Yaskawa INFORM job: DEMO_ROOF_UPPER_0625_3PAINT_26.JBI

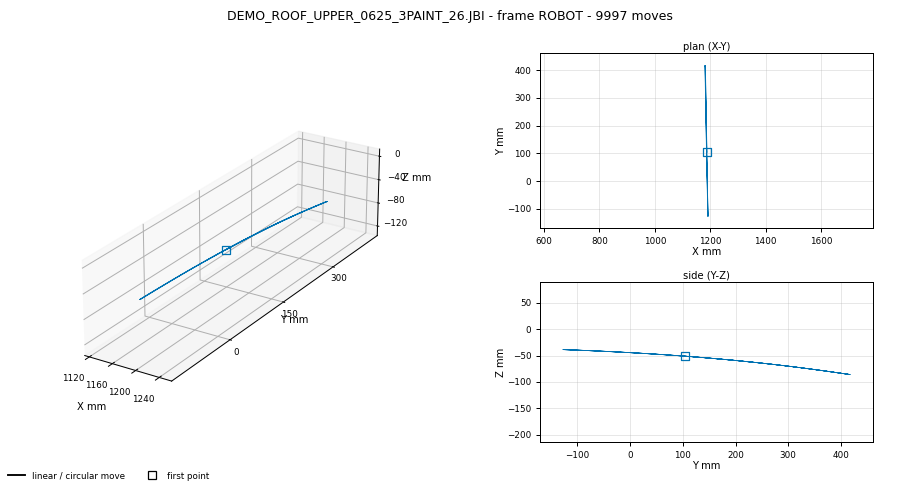
[picture p0: tool path of DEMO_ROOF_UPPER_0625_3PAINT_26.JBI in frame ROBOT, 9997 of 9997 moves have a stored position in this frame; points joined in program order, loops and branches not executed]
/JOB
//NAME DEMO_ROOF_UPPER_0625_3PAINT26
//POS
///NPOS 9997,0,0,0,0,0
///TOOL 0
///USER 0
///POSTYPE ROBOT
///RECTAN
///RCONF 1,0,0,0,0,0,0,0,0,0,0,0,0,0,0,0,0,0,0,0,0,0,0,0
C00000=1188.061,103.927,-51.027,-178.803,6.071,148.735
C00001=1188.057,104.176,-51.046,-178.800,6.072,148.734
C00002=1188.052,104.425,-51.064,-178.798,6.073,148.734
C00003=1188.047,104.675,-51.083,-178.795,6.075,148.733
C00004=1188.042,104.924,-51.102,-178.793,6.076,148.733
C00005=1188.036,105.173,-51.120,-178.790,6.077,148.732
C00006=1188.032,105.423,-51.139,-178.787,6.078,148.732
C00007=1188.027,105.672,-51.157,-178.785,6.080,148.731
C00008=1188.023,105.921,-51.177,-178.782,6.080,148.731
C00009=1188.018,106.171,-51.195,-178.779,6.082,148.730
C00010=1188.012,106.439,-51.216,-178.776,6.083,148.730
C00011=1188.008,106.708,-51.236,-178.774,6.084,148.729
C00012=1188.002,106.975,-51.256,-178.771,6.086,148.729
C00013=1187.996,107.244,-51.276,-178.768,6.087,148.728
C00014=1187.992,107.493,-51.295,-178.766,6.088,148.728
C00015=1187.987,107.743,-51.314,-178.763,6.090,148.727
C00016=1187.983,107.992,-51.333,-178.760,6.090,148.727
C00017=1187.978,108.241,-51.351,-178.758,6.092,148.726
C00018=1187.973,108.490,-51.370,-178.755,6.094,148.726
C00019=1187.969,108.739,-51.389,-178.752,6.094,148.725
C00020=1187.963,108.989,-51.408,-178.750,6.096,148.725
C00021=1187.959,109.238,-51.427,-178.747,6.097,148.724
C00022=1187.954,109.487,-51.446,-178.744,6.098,148.724
C00023=1187.949,109.736,-51.464,-178.742,6.099,148.723
C00024=1187.944,109.986,-51.484,-178.739,6.101,148.723
C00025=1187.939,110.234,-51.503,-178.737,6.102,148.722
C00026=1187.934,110.484,-51.521,-178.734,6.103,148.722
C00027=1187.929,110.733,-51.541,-178.731,6.105,148.721
C00028=1187.925,110.983,-51.560,-178.729,6.106,148.721
C00029=1187.919,111.232,-51.578,-178.726,6.107,148.720
C00030=1187.915,111.481,-51.597,-178.723,6.108,148.720
C00031=1187.910,111.730,-51.617,-178.721,6.110,148.719
C00032=1187.906,111.979,-51.636,-178.718,6.110,148.719
C00033=1187.900,112.229,-51.654,-178.715,6.112,148.718
C00034=1187.896,112.478,-51.673,-178.712,6.113,148.718
C00035=1187.891,112.727,-51.693,-178.710,6.114,148.717
C00036=1187.886,112.977,-51.712,-178.707,6.116,148.717
C00037=1187.881,113.226,-51.730,-178.705,6.117,148.716
C00038=1187.877,113.475,-51.750,-178.702,6.118,148.716
C00039=1187.871,113.724,-51.769,-178.700,6.119,148.715
C00040=1187.867,113.973,-51.788,-178.697,6.121,148.715
C00041=1187.862,114.222,-51.808,-178.694,6.122,148.714
C00042=1187.857,114.472,-51.826,-178.691,6.123,148.714
C00043=1187.852,114.721,-51.845,-178.689,6.125,148.713
C00044=1187.847,114.971,-51.865,-178.687,6.126,148.713
C00045=1187.843,115.219,-51.884,-178.683,6.127,148.712
C00046=1187.838,115.469,-51.903,-178.681,6.129,148.712
C00047=1187.833,115.718,-51.923,-178.679,6.130,148.712
C00048=1187.829,115.967,-51.942,-178.675,6.131,148.711
C00049=1187.823,116.216,-51.961,-178.673,6.132,148.710
C00050=1187.819,116.465,-51.981,-178.671,6.134,148.710
C00051=1187.813,116.714,-52.000,-178.667,6.135,148.709
C00052=1187.809,116.964,-52.018,-178.665,6.136,148.709
C00053=1187.804,117.214,-52.038,-178.663,6.138,148.709
C00054=1187.799,117.462,-52.057,-178.660,6.138,148.708
C00055=1187.795,117.712,-52.076,-178.657,6.140,148.708
C00056=1187.790,117.961,-52.096,-178.655,6.142,148.707
C00057=1187.785,118.210,-52.115,-178.652,6.142,148.707
C00058=1187.780,118.460,-52.135,-178.649,6.144,148.706
C00059=1187.775,118.708,-52.154,-178.647,6.145,148.706
C00060=1187.771,118.958,-52.173,-178.644,6.147,148.705
C00061=1187.765,119.207,-52.192,-178.641,6.148,148.705
C00062=1187.761,119.456,-52.212,-178.639,6.149,148.704
C00063=1187.756,119.706,-52.232,-178.636,6.151,148.704
C00064=1187.752,119.954,-52.251,-178.633,6.152,148.703
C00065=1187.747,120.203,-52.271,-178.631,6.153,148.703
C00066=1187.741,120.452,-52.290,-178.628,6.155,148.702
C00067=1187.737,120.702,-52.310,-178.626,6.156,148.702
C00068=1187.732,120.951,-52.329,-178.623,6.157,148.701
C00069=1187.727,121.200,-52.348,-178.620,6.159,148.701
C00070=1187.723,121.450,-52.368,-178.618,6.160,148.700
C00071=1187.718,121.699,-52.387,-178.615,6.161,148.700
C00072=1187.713,121.948,-52.407,-178.612,6.163,148.699
C00073=1187.708,122.197,-52.427,-178.610,6.164,148.699
C00074=1187.703,122.446,-52.447,-178.607,6.166,148.699
C00075=1187.698,122.695,-52.466,-178.604,6.166,148.698
C00076=1187.694,122.945,-52.485,-178.602,6.168,148.698
C00077=1187.689,123.194,-52.505,-178.599,6.170,148.697
C00078=1187.684,123.443,-52.524,-178.596,6.170,148.697
C00079=1187.680,123.692,-52.544,-178.594,6.172,148.696
C00080=1187.675,123.942,-52.564,-178.591,6.174,148.696
C00081=1187.669,124.190,-52.583,-178.588,6.174,148.695
C00082=1187.665,124.440,-52.603,-178.586,6.176,148.695
C00083=1187.660,124.689,-52.623,-178.583,6.178,148.694
C00084=1187.655,124.938,-52.643,-178.581,6.179,148.694
C00085=1187.650,125.187,-52.662,-178.578,6.180,148.693
C00086=1187.646,125.437,-52.681,-178.575,6.182,148.693
C00087=1187.642,125.686,-52.702,-178.573,6.183,148.692
C00088=1187.636,125.934,-52.721,-178.570,6.184,148.692
C00089=1187.632,126.184,-52.741,-178.567,6.186,148.691
C00090=1187.627,126.433,-52.761,-178.565,6.187,148.691
C00091=1187.622,126.683,-52.781,-178.562,6.188,148.690
C00092=1187.617,126.931,-52.800,-178.559,6.190,148.690
C00093=1187.613,127.180,-52.820,-178.557,6.191,148.690
C00094=1187.608,127.430,-52.840,-178.554,6.193,148.689
C00095=1187.603,127.679,-52.860,-178.551,6.194,148.689
C00096=1187.598,127.928,-52.880,-178.549,6.195,148.688
C00097=1187.593,128.177,-52.899,-178.546,6.197,148.688
C00098=1187.589,128.426,-52.920,-178.543,6.198,148.687
C00099=1187.584,128.676,-52.939,-178.541,6.199,148.687
C00100=1187.579,128.924,-52.959,-178.538,6.201,148.686
C00101=1187.574,129.174,-52.979,-178.536,6.203,148.686
C00102=1187.570,129.423,-52.999,-178.533,6.203,148.685
C00103=1187.565,129.672,-53.020,-178.530,6.205,148.685
C00104=1187.560,129.922,-53.039,-178.528,6.207,148.685
C00105=1187.555,130.170,-53.059,-178.525,6.208,148.684
C00106=1187.550,130.420,-53.079,-178.522,6.209,148.684
C00107=1187.546,130.669,-53.099,-178.520,6.211,148.683
C00108=1187.541,130.918,-53.119,-178.517,6.213,148.683
C00109=1187.536,131.167,-53.139,-178.514,6.213,148.682
C00110=1187.531,131.416,-53.159,-178.512,6.215,148.682
C00111=1187.527,131.665,-53.179,-178.509,6.217,148.681
C00112=1187.522,131.915,-53.199,-178.507,6.218,148.681
C00113=1187.517,132.164,-53.220,-178.504,6.219,148.680
C00114=1187.512,132.433,-53.241,-178.501,6.221,148.680
C00115=1187.506,132.701,-53.263,-178.498,6.223,148.680
C00116=1187.502,132.970,-53.284,-178.495,6.224,148.679
C00117=1187.496,133.238,-53.307,-178.492,6.226,148.679
C00118=1187.491,133.488,-53.326,-178.490,6.226,148.678
C00119=1187.487,133.736,-53.347,-178.487,6.228,148.678
C00120=1187.482,133.986,-53.366,-178.484,6.230,148.677
C00121=1187.478,134.235,-53.387,-178.482,6.232,148.677
C00122=1187.472,134.484,-53.407,-178.479,6.232,148.676
C00123=1187.467,134.733,-53.427,-178.476,6.234,148.676
C00124=1187.463,134.982,-53.447,-178.474,6.236,148.675
C00125=1187.458,135.231,-53.468,-178.472,6.237,148.675
C00126=1187.454,135.480,-53.488,-178.468,6.238,148.674
C00127=1187.448,135.730,-53.508,-178.466,6.240,148.674
C00128=1187.444,135.979,-53.529,-178.463,6.242,148.674
C00129=1187.440,136.228,-53.549,-178.461,6.242,148.673
C00130=1187.435,136.477,-53.569,-178.458,6.244,148.673
C00131=1187.430,136.727,-53.590,-178.455,6.246,148.672
C00132=1187.425,136.976,-53.610,-178.452,6.247,148.672
C00133=1187.420,137.224,-53.630,-178.450,6.248,148.671
C00134=1187.415,137.473,-53.650,-178.447,6.250,148.671
C00135=1187.410,137.723,-53.671,-178.444,6.252,148.670
C00136=1187.406,137.972,-53.691,-178.442,6.252,148.670
C00137=1187.401,138.220,-53.712,-178.440,6.254,148.670
C00138=1187.396,138.470,-53.732,-178.437,6.256,148.669
C00139=1187.392,138.719,-53.753,-178.434,6.257,148.669
C00140=1187.387,138.968,-53.773,-178.432,6.258,148.668
C00141=1187.382,139.218,-53.793,-178.429,6.260,148.668
C00142=1187.377,139.466,-53.814,-178.426,6.262,148.667
C00143=1187.373,139.715,-53.834,-178.423,6.264,148.667
C00144=1187.368,139.965,-53.855,-178.421,6.264,148.666
C00145=1187.363,140.214,-53.876,-178.418,6.266,148.666
C00146=1187.359,140.463,-53.896,-178.415,6.268,148.666
C00147=1187.354,140.712,-53.917,-178.413,6.270,148.665
C00148=1187.349,140.961,-53.937,-178.410,6.271,148.665
C00149=1187.344,141.211,-53.958,-178.407,6.272,148.664
C00150=1187.339,141.460,-53.978,-178.405,6.274,148.664
C00151=1187.335,141.709,-53.998,-178.402,6.275,148.664
C00152=1187.330,141.958,-54.019,-178.399,6.277,148.663
C00153=1187.325,142.207,-54.040,-178.397,6.278,148.663
C00154=1187.320,142.456,-54.061,-178.394,6.280,148.662
C00155=1187.316,142.705,-54.081,-178.391,6.281,148.662
C00156=1187.311,142.954,-54.101,-178.389,6.283,148.661
C00157=1187.306,143.203,-54.122,-178.387,6.284,148.661
C00158=1187.302,143.452,-54.143,-178.384,6.286,148.661
C00159=1187.297,143.701,-54.164,-178.381,6.287,148.660
C00160=1187.292,143.950,-54.184,-178.378,6.289,148.660
C00161=1187.287,144.199,-54.206,-178.375,6.291,148.659
C00162=1187.283,144.448,-54.226,-178.373,6.292,148.659
C00163=1187.278,144.697,-54.247,-178.371,6.293,148.658
C00164=1187.274,144.947,-54.268,-178.367,6.295,148.658
C00165=1187.269,145.196,-54.289,-178.365,6.297,148.657
C00166=1187.264,145.445,-54.309,-178.363,6.298,148.657
C00167=1187.259,145.694,-54.330,-178.360,6.299,148.657
C00168=1187.255,145.943,-54.350,-178.357,6.301,148.656
C00169=1187.249,146.193,-54.371,-178.355,6.303,148.656
C00170=1187.245,146.441,-54.392,-178.351,6.304,148.655
C00171=1187.240,146.690,-54.413,-178.349,6.305,148.655
C00172=1187.236,146.939,-54.434,-178.347,6.307,148.655
C00173=1187.230,147.188,-54.455,-178.344,6.309,148.654
C00174=1187.225,147.438,-54.476,-178.341,6.310,148.654
C00175=1187.222,147.687,-54.497,-178.339,6.312,148.653
C00176=1187.217,147.936,-54.518,-178.335,6.314,148.653
C00177=1187.212,148.185,-54.539,-178.333,6.315,148.652
C00178=1187.207,148.434,-54.560,-178.331,6.316,148.652
C00179=1187.203,148.682,-54.581,-178.328,6.318,148.652
C00180=1187.198,148.932,-54.602,-178.325,6.320,148.651
C00181=1187.193,149.181,-54.623,-178.322,6.322,148.651
C00182=1187.189,149.431,-54.643,-178.320,6.322,148.650
C00183=1187.184,149.679,-54.665,-178.317,6.324,148.650
C00184=1187.179,149.928,-54.686,-178.315,6.326,148.649
C00185=1187.174,150.177,-54.706,-178.312,6.328,148.649
C00186=1187.169,150.426,-54.728,-178.309,6.329,148.649
C00187=1187.164,150.675,-54.749,-178.306,6.331,148.648
C00188=1187.160,150.925,-54.770,-178.304,6.332,148.648
C00189=1187.155,151.174,-54.791,-178.301,6.334,148.647
C00190=1187.150,151.423,-54.812,-178.299,6.335,148.647
C00191=1187.146,151.672,-54.833,-178.296,6.337,148.647
C00192=1187.141,151.920,-54.854,-178.293,6.339,148.646
C00193=1187.136,152.170,-54.875,-178.291,6.340,148.646
C00194=1187.132,152.419,-54.897,-178.288,6.342,148.645
C00195=1187.127,152.668,-54.918,-178.286,6.343,148.645
C00196=1187.122,152.917,-54.939,-178.283,6.345,148.645
C00197=1187.117,153.166,-54.960,-178.280,6.347,148.644
C00198=1187.113,153.416,-54.981,-178.277,6.348,148.644
C00199=1187.108,153.664,-55.003,-178.274,6.350,148.643
C00200=1187.103,153.913,-55.024,-178.272,6.351,148.643
C00201=1187.098,154.162,-55.045,-178.270,6.353,148.643
C00202=1187.094,154.411,-55.066,-178.267,6.355,148.642
C00203=1187.090,154.660,-55.088,-178.264,6.356,148.642
C00204=1187.084,154.910,-55.109,-178.262,6.358,148.641
C00205=1187.080,155.158,-55.131,-178.258,6.360,148.641
C00206=1187.074,155.408,-55.152,-178.256,6.361,148.640
C00207=1187.071,155.657,-55.173,-178.254,6.362,148.640
C00208=1187.066,155.906,-55.194,-178.251,6.364,148.640
C00209=1187.061,156.154,-55.216,-178.248,6.366,148.639
C00210=1187.057,156.404,-55.238,-178.246,6.368,148.639
C00211=1187.051,156.653,-55.259,-178.243,6.369,148.639
C00212=1187.046,156.902,-55.280,-178.240,6.371,148.638
C00213=1187.042,157.151,-55.301,-178.238,6.373,148.638
C00214=1187.038,157.400,-55.323,-178.235,6.373,148.637
C00215=1187.033,157.649,-55.344,-178.232,6.375,148.637
C00216=1187.028,157.898,-55.365,-178.230,6.377,148.636
C00217=1187.023,158.147,-55.387,-178.227,6.379,148.636
C00218=1187.019,158.416,-55.410,-178.224,6.381,148.636
C00219=1187.013,158.684,-55.434,-178.222,6.382,148.635
C00220=1187.008,158.953,-55.457,-178.218,6.384,148.635
C00221=1187.003,159.223,-55.480,-178.215,6.386,148.634
C00222=1186.998,159.472,-55.502,-178.213,6.387,148.634
C00223=1186.994,159.721,-55.524,-178.210,6.389,148.634
C00224=1186.988,159.970,-55.545,-178.208,6.391,148.633
C00225=1186.984,160.219,-55.567,-178.205,6.393,148.633
C00226=1186.979,160.468,-55.588,-178.202,6.394,148.633
C00227=1186.975,160.716,-55.610,-178.200,6.396,148.632
C00228=1186.971,160.966,-55.631,-178.197,6.398,148.632
C00229=1186.966,161.215,-55.653,-178.194,6.400,148.631
C00230=1186.961,161.464,-55.675,-178.191,6.401,148.631
C00231=1186.957,161.713,-55.696,-178.189,6.402,148.630
C00232=1186.952,161.962,-55.718,-178.186,6.404,148.630
C00233=1186.947,162.211,-55.739,-178.184,6.406,148.630
C00234=1186.942,162.460,-55.761,-178.181,6.407,148.629
C00235=1186.938,162.709,-55.783,-178.178,6.409,148.629
C00236=1186.933,162.958,-55.805,-178.176,6.411,148.629
C00237=1186.928,163.207,-55.826,-178.173,6.413,148.628
C00238=1186.924,163.456,-55.848,-178.170,6.415,148.628
C00239=1186.919,163.705,-55.870,-178.168,6.416,148.627
C00240=1186.915,163.954,-55.892,-178.165,6.418,148.627
C00241=1186.909,164.204,-55.914,-178.162,6.420,148.627
C00242=1186.904,164.452,-55.935,-178.159,6.422,148.626
C00243=1186.900,164.702,-55.957,-178.157,6.423,148.626
C00244=1186.895,164.950,-55.979,-178.155,6.424,148.626
C00245=1186.891,165.200,-56.001,-178.152,6.426,148.625
C00246=1186.886,165.448,-56.023,-178.149,6.428,148.625
C00247=1186.881,165.698,-56.045,-178.146,6.429,148.624
C00248=1186.877,165.946,-56.067,-178.144,6.431,148.624
C00249=1186.872,166.196,-56.089,-178.141,6.433,148.624
C00250=1186.867,166.444,-56.110,-178.138,6.435,148.623
C00251=1186.863,166.694,-56.132,-178.135,6.437,148.623
C00252=1186.858,166.942,-56.155,-178.133,6.438,148.622
C00253=1186.853,167.191,-56.176,-178.130,6.440,148.622
C00254=1186.848,167.440,-56.198,-178.127,6.442,148.622
C00255=1186.844,167.688,-56.221,-178.125,6.444,148.621
C00256=1186.840,167.938,-56.243,-178.122,6.445,148.621
C00257=1186.835,168.186,-56.265,-178.119,6.447,148.621
C00258=1186.830,168.436,-56.287,-178.117,6.448,148.620
C00259=1186.825,168.685,-56.309,-178.115,6.450,148.620
C00260=1186.821,168.934,-56.331,-178.112,6.452,148.619
C00261=1186.816,169.183,-56.353,-178.109,6.453,148.619
C00262=1186.812,169.432,-56.375,-178.107,6.455,148.619
C00263=1186.806,169.681,-56.397,-178.104,6.457,148.618
C00264=1186.802,169.930,-56.420,-178.101,6.459,148.618
C00265=1186.798,170.179,-56.442,-178.099,6.461,148.618
C00266=1186.793,170.428,-56.463,-178.096,6.462,148.617
C00267=1186.788,170.677,-56.486,-178.093,6.464,148.617
C00268=1186.783,170.926,-56.508,-178.091,6.466,148.617
C00269=1186.779,171.175,-56.531,-178.088,6.468,148.616
C00270=1186.774,171.423,-56.552,-178.085,6.470,148.616
C00271=1186.769,171.673,-56.575,-178.083,6.471,148.615
C00272=1186.764,171.922,-56.597,-178.080,6.473,148.615
C00273=1186.760,172.170,-56.619,-178.077,6.475,148.615
C00274=1186.755,172.420,-56.642,-178.074,6.477,148.614
C00275=1186.750,172.669,-56.664,-178.072,6.478,148.614
C00276=1186.746,172.917,-56.686,-178.069,6.480,148.614
C00277=1186.742,173.166,-56.708,-178.066,6.482,148.613
C00278=1186.737,173.416,-56.731,-178.064,6.484,148.613
C00279=1186.732,173.664,-56.753,-178.061,6.486,148.613
C00280=1186.728,173.913,-56.775,-178.058,6.487,148.612
C00281=1186.723,174.163,-56.798,-178.056,6.489,148.612
C00282=1186.718,174.411,-56.820,-178.053,6.491,148.611
C00283=1186.713,174.660,-56.843,-178.050,6.493,148.611
C00284=1186.709,174.910,-56.865,-178.048,6.494,148.611
C00285=1186.704,175.158,-56.887,-178.045,6.496,148.610
C00286=1186.699,175.407,-56.910,-178.042,6.498,148.610
C00287=1186.695,175.655,-56.932,-178.040,6.500,148.610
C00288=1186.690,175.905,-56.954,-178.037,6.502,148.609
C00289=1186.685,176.154,-56.977,-178.034,6.503,148.609
C00290=1186.681,176.402,-56.999,-178.032,6.505,148.609
C00291=1186.676,176.652,-57.022,-178.029,6.507,148.608
C00292=1186.672,176.901,-57.045,-178.026,6.509,148.608
C00293=1186.666,177.150,-57.067,-178.024,6.511,148.607
C00294=1186.662,177.398,-57.090,-178.021,6.512,148.607
C00295=1186.657,177.648,-57.112,-178.018,6.514,148.607
C00296=1186.653,177.896,-57.135,-178.016,6.516,148.606
C00297=1186.649,178.145,-57.157,-178.013,6.518,148.606
C00298=1186.644,178.395,-57.180,-178.010,6.519,148.606
C00299=1186.639,178.643,-57.203,-178.008,6.522,148.606
C00300=1186.634,178.892,-57.225,-178.005,6.523,148.605
C00301=1186.630,179.141,-57.248,-178.003,6.525,148.605
C00302=1186.625,179.391,-57.271,-178.000,6.527,148.604
C00303=1186.621,179.639,-57.293,-177.997,6.529,148.604
C00304=1186.616,179.888,-57.317,-177.995,6.531,148.604
C00305=1186.612,180.137,-57.339,-177.992,6.532,148.603
C00306=1186.606,180.385,-57.362,-177.989,6.534,148.603
C00307=1186.602,180.635,-57.384,-177.987,6.536,148.603
C00308=1186.597,180.884,-57.407,-177.984,6.538,148.602
C00309=1186.593,181.133,-57.430,-177.981,6.539,148.602
C00310=1186.588,181.381,-57.452,-177.979,6.541,148.602
C00311=1186.583,181.630,-57.475,-177.976,6.543,148.601
C00312=1186.579,181.879,-57.498,-177.973,6.545,148.601
C00313=1186.575,182.128,-57.521,-177.971,6.547,148.600
C00314=1186.570,182.377,-57.543,-177.968,6.548,148.600
C00315=1186.565,182.626,-57.567,-177.965,6.550,148.600
C00316=1186.560,182.875,-57.590,-177.963,6.552,148.600
C00317=1186.556,183.124,-57.613,-177.961,6.554,148.599
C00318=1186.551,183.373,-57.635,-177.958,6.556,148.599
C00319=1186.546,183.622,-57.658,-177.955,6.558,148.599
C00320=1186.542,183.870,-57.681,-177.952,6.560,148.598
C00321=1186.537,184.119,-57.704,-177.949,6.562,148.598
C00322=1186.533,184.389,-57.729,-177.947,6.564,148.598
C00323=1186.527,184.659,-57.754,-177.944,6.566,148.597
C00324=1186.522,184.928,-57.779,-177.941,6.568,148.597
C00325=1186.518,185.198,-57.803,-177.938,6.570,148.596
C00326=1186.513,185.447,-57.827,-177.935,6.572,148.596
C00327=1186.508,185.696,-57.850,-177.933,6.574,148.596
C00328=1186.504,185.945,-57.873,-177.930,6.575,148.595
C00329=1186.499,186.193,-57.896,-177.927,6.577,148.595
C00330=1186.494,186.443,-57.918,-177.925,6.579,148.595
C00331=1186.489,186.692,-57.942,-177.922,6.581,148.594
C00332=1186.485,186.940,-57.965,-177.919,6.583,148.594
C00333=1186.481,187.189,-57.988,-177.917,6.584,148.594
C00334=1186.476,187.438,-58.011,-177.914,6.587,148.594
C00335=1186.471,187.687,-58.034,-177.911,6.589,148.593
C00336=1186.467,187.935,-58.057,-177.909,6.591,148.593
C00337=1186.462,188.184,-58.080,-177.906,6.593,148.592
C00338=1186.457,188.433,-58.104,-177.903,6.595,148.592
C00339=1186.452,188.682,-58.127,-177.901,6.596,148.592
C00340=1186.449,188.931,-58.150,-177.898,6.598,148.591
C00341=1186.444,189.180,-58.173,-177.895,6.600,148.591
C00342=1186.439,189.429,-58.197,-177.893,6.602,148.591
C00343=1186.434,189.678,-58.220,-177.890,6.604,148.591
C00344=1186.429,189.927,-58.243,-177.888,6.606,148.590
C00345=1186.424,190.176,-58.266,-177.885,6.607,148.590
C00346=1186.420,190.424,-58.289,-177.882,6.610,148.590
C00347=1186.416,190.673,-58.313,-177.879,6.612,148.589
C00348=1186.411,190.922,-58.337,-177.877,6.614,148.589
C00349=1186.407,191.171,-58.360,-177.874,6.615,148.588
C00350=1186.402,191.420,-58.383,-177.872,6.618,148.588
C00351=1186.397,191.669,-58.407,-177.869,6.619,148.588
C00352=1186.393,191.918,-58.430,-177.866,6.621,148.588
C00353=1186.388,192.167,-58.453,-177.864,6.623,148.587
C00354=1186.384,192.415,-58.477,-177.861,6.625,148.587
C00355=1186.379,192.664,-58.500,-177.858,6.627,148.587
C00356=1186.375,192.913,-58.524,-177.855,6.629,148.586
C00357=1186.370,193.162,-58.547,-177.853,6.631,148.586
C00358=1186.365,193.411,-58.570,-177.850,6.633,148.586
C00359=1186.361,193.660,-58.594,-177.848,6.635,148.585
C00360=1186.356,193.909,-58.618,-177.845,6.637,148.585
C00361=1186.352,194.158,-58.641,-177.842,6.638,148.585
C00362=1186.347,194.407,-58.664,-177.840,6.640,148.584
C00363=1186.343,194.655,-58.688,-177.836,6.643,148.584
C00364=1186.338,194.904,-58.712,-177.834,6.645,148.584
C00365=1186.333,195.153,-58.735,-177.832,6.647,148.584
C00366=1186.329,195.402,-58.759,-177.829,6.649,148.583
C00367=1186.324,195.651,-58.783,-177.826,6.650,148.583
C00368=1186.319,195.900,-58.806,-177.824,6.652,148.583
C00369=1186.315,196.148,-58.830,-177.821,6.654,148.582
C00370=1186.310,196.397,-58.853,-177.819,6.656,148.582
C00371=1186.306,196.646,-58.877,-177.815,6.659,148.582
C00372=1186.301,196.895,-58.901,-177.813,6.661,148.581
C00373=1186.296,197.144,-58.924,-177.810,6.662,148.581
C00374=1186.292,197.392,-58.948,-177.807,6.664,148.581
C00375=1186.287,197.641,-58.972,-177.805,6.666,148.581
C00376=1186.283,197.890,-58.995,-177.803,6.668,148.580
C00377=1186.278,198.138,-59.019,-177.800,6.670,148.580
C00378=1186.274,198.388,-59.042,-177.797,6.672,148.580
C00379=1186.269,198.636,-59.067,-177.794,6.674,148.579
C00380=1186.264,198.885,-59.090,-177.791,6.676,148.579
C00381=1186.259,199.134,-59.115,-177.789,6.678,148.579
C00382=1186.255,199.383,-59.138,-177.787,6.680,148.578
C00383=1186.250,199.631,-59.162,-177.784,6.682,148.578
C00384=1186.246,199.881,-59.186,-177.781,6.684,148.578
C00385=1186.242,200.129,-59.210,-177.778,6.686,148.577
C00386=1186.237,200.378,-59.233,-177.776,6.688,148.577
C00387=1186.233,200.627,-59.257,-177.773,6.690,148.577
C00388=1186.227,200.876,-59.281,-177.770,6.692,148.577
C00389=1186.223,201.124,-59.305,-177.768,6.694,148.576
C00390=1186.218,201.373,-59.329,-177.765,6.696,148.576
C00391=1186.214,201.622,-59.353,-177.762,6.699,148.576
C00392=1186.210,201.871,-59.377,-177.760,6.700,148.575
C00393=1186.204,202.120,-59.401,-177.757,6.702,148.575
C00394=1186.200,202.369,-59.425,-177.754,6.704,148.575
C00395=1186.196,202.617,-59.449,-177.752,6.707,148.575
C00396=1186.191,202.866,-59.473,-177.749,6.709,148.574
C00397=1186.187,203.115,-59.497,-177.746,6.711,148.574
C00398=1186.181,203.363,-59.521,-177.744,6.712,148.574
C00399=1186.177,203.613,-59.545,-177.741,6.714,148.573
C00400=1186.173,203.862,-59.569,-177.739,6.716,148.573
C00401=1186.169,204.110,-59.593,-177.736,6.719,148.573
C00402=1186.163,204.359,-59.618,-177.733,6.721,148.573
C00403=1186.159,204.608,-59.641,-177.730,6.722,148.572
C00404=1186.155,204.857,-59.666,-177.728,6.725,148.572
C00405=1186.151,205.105,-59.690,-177.725,6.726,148.572
C00406=1186.145,205.354,-59.714,-177.722,6.729,148.571
C00407=1186.141,205.603,-59.738,-177.720,6.731,148.571
C00408=1186.136,205.851,-59.762,-177.717,6.733,148.571
C00409=1186.132,206.101,-59.787,-177.715,6.735,148.571
C00410=1186.127,206.349,-59.811,-177.712,6.737,148.570
C00411=1186.123,206.598,-59.835,-177.709,6.739,148.570
C00412=1186.118,206.847,-59.859,-177.707,6.741,148.570
C00413=1186.114,207.096,-59.883,-177.704,6.743,148.569
C00414=1186.109,207.345,-59.907,-177.701,6.745,148.569
C00415=1186.104,207.593,-59.932,-177.698,6.748,148.569
C00416=1186.100,207.842,-59.956,-177.696,6.750,148.569
C00417=1186.095,208.091,-59.981,-177.693,6.752,148.568
C00418=1186.091,208.339,-60.005,-177.691,6.753,148.568
C00419=1186.087,208.588,-60.029,-177.688,6.755,148.568
C00420=1186.081,208.837,-60.054,-177.685,6.758,148.568
C00421=1186.078,209.086,-60.079,-177.683,6.760,148.567
C00422=1186.072,209.335,-60.102,-177.680,6.762,148.567
C00423=1186.068,209.583,-60.127,-177.677,6.764,148.567
C00424=1186.063,209.832,-60.151,-177.674,6.766,148.566
C00425=1186.059,210.081,-60.176,-177.672,6.768,148.566
C00426=1186.054,210.351,-60.202,-177.669,6.770,148.566
C00427=1186.049,210.622,-60.229,-177.666,6.773,148.565
C00428=1186.044,210.893,-60.256,-177.663,6.775,148.565
C00429=1186.040,211.162,-60.282,-177.660,6.777,148.565
C00430=1186.034,211.411,-60.307,-177.658,6.779,148.565
C00431=1186.030,211.660,-60.331,-177.655,6.781,148.564
C00432=1186.026,211.909,-60.356,-177.652,6.784,148.564
C00433=1186.021,212.157,-60.380,-177.650,6.786,148.564
C00434=1186.016,212.406,-60.405,-177.647,6.788,148.564
C00435=1186.011,212.656,-60.430,-177.645,6.789,148.563
C00436=1186.007,212.904,-60.454,-177.641,6.792,148.563
C00437=1186.003,213.153,-60.479,-177.639,6.794,148.563
C00438=1185.998,213.401,-60.504,-177.636,6.796,148.563
C00439=1185.993,213.650,-60.528,-177.634,6.798,148.562
C00440=1185.990,213.899,-60.553,-177.631,6.801,148.562
C00441=1185.984,214.148,-60.578,-177.628,6.803,148.562
C00442=1185.980,214.396,-60.602,-177.626,6.804,148.561
C00443=1185.976,214.645,-60.627,-177.624,6.807,148.561
C00444=1185.971,214.894,-60.652,-177.620,6.809,148.561
C00445=1185.967,215.143,-60.676,-177.618,6.811,148.561
C00446=1185.962,215.391,-60.701,-177.616,6.813,148.561
C00447=1185.958,215.639,-60.726,-177.612,6.816,148.560
C00448=1185.953,215.889,-60.751,-177.610,6.818,148.560
C00449=1185.948,216.137,-60.776,-177.607,6.819,148.560
C00450=1185.944,216.387,-60.800,-177.605,6.822,148.559
C00451=1185.939,216.635,-60.825,-177.602,6.824,148.559
C00452=1185.934,216.883,-60.850,-177.599,6.826,148.559
C00453=1185.930,217.132,-60.875,-177.597,6.828,148.559
C00454=1185.926,217.381,-60.900,-177.594,6.831,148.558
C00455=1185.921,217.630,-60.925,-177.591,6.833,148.558
C00456=1185.917,217.878,-60.949,-177.589,6.835,148.558
C00457=1185.912,218.127,-60.975,-177.586,6.837,148.558
C00458=1185.907,218.376,-60.999,-177.583,6.839,148.557
C00459=1185.904,218.625,-61.024,-177.581,6.841,148.557
C00460=1185.899,218.873,-61.049,-177.578,6.843,148.557
C00461=1185.894,219.123,-61.074,-177.575,6.846,148.557
C00462=1185.889,219.371,-61.100,-177.573,6.848,148.556
C00463=1185.885,219.619,-61.124,-177.570,6.850,148.556
C00464=1185.881,219.868,-61.150,-177.568,6.852,148.556
C00465=1185.876,220.117,-61.174,-177.565,6.855,148.556
C00466=1185.871,220.365,-61.200,-177.562,6.856,148.555
C00467=1185.867,220.614,-61.224,-177.560,6.858,148.555
C00468=1185.863,220.863,-61.250,-177.557,6.861,148.555
C00469=1185.858,221.111,-61.274,-177.554,6.863,148.555
C00470=1185.853,221.360,-61.300,-177.552,6.865,148.555
C00471=1185.850,221.609,-61.325,-177.548,6.868,148.554
C00472=1185.845,221.857,-61.350,-177.546,6.870,148.554
C00473=1185.840,222.107,-61.375,-177.544,6.872,148.554
C00474=1185.835,222.355,-61.400,-177.541,6.873,148.553
C00475=1185.831,222.604,-61.425,-177.538,6.876,148.553
C00476=1185.826,222.852,-61.451,-177.536,6.878,148.553
C00477=1185.822,223.101,-61.477,-177.533,6.880,148.553
C00478=1185.817,223.350,-61.501,-177.530,6.883,148.553
C00479=1185.813,223.598,-61.526,-177.528,6.885,148.552
C00480=1185.808,223.847,-61.552,-177.525,6.887,148.552
C00481=1185.804,224.096,-61.577,-177.522,6.890,148.552
C00482=1185.800,224.345,-61.603,-177.520,6.891,148.552
C00483=1185.795,224.593,-61.628,-177.517,6.894,148.551
C00484=1185.790,224.842,-61.653,-177.514,6.896,148.551
C00485=1185.785,225.090,-61.678,-177.511,6.898,148.551
C00486=1185.781,225.339,-61.704,-177.509,6.900,148.551
C00487=1185.777,225.588,-61.728,-177.506,6.903,148.550
C00488=1185.773,225.836,-61.754,-177.504,6.905,148.550
C00489=1185.768,226.085,-61.780,-177.501,6.907,148.550
C00490=1185.764,226.333,-61.805,-177.498,6.910,148.550
C00491=1185.759,226.583,-61.830,-177.496,6.912,148.550
C00492=1185.755,226.832,-61.856,-177.493,6.913,148.549
C00493=1185.750,227.080,-61.881,-177.490,6.916,148.549
C00494=1185.746,227.329,-61.907,-177.488,6.918,148.549
C00495=1185.741,227.577,-61.932,-177.486,6.920,148.549
C00496=1185.736,227.826,-61.957,-177.482,6.923,148.548
C00497=1185.732,228.075,-61.983,-177.480,6.925,148.548
C00498=1185.727,228.323,-62.009,-177.478,6.927,148.548
C00499=1185.723,228.572,-62.034,-177.474,6.930,148.548
C00500=1185.719,228.821,-62.060,-177.472,6.932,148.548
C00501=1185.714,229.069,-62.085,-177.469,6.934,148.547
C00502=1185.710,229.317,-62.111,-177.467,6.937,148.547
C00503=1185.706,229.566,-62.137,-177.464,6.938,148.547
C00504=1185.700,229.815,-62.163,-177.461,6.941,148.547
C00505=1185.696,230.064,-62.188,-177.459,6.943,148.546
C00506=1185.691,230.313,-62.214,-177.456,6.945,148.546
C00507=1185.686,230.561,-62.239,-177.453,6.948,148.546
C00508=1185.682,230.810,-62.265,-177.451,6.950,148.546
C00509=1185.678,231.059,-62.291,-177.449,6.952,148.546
C00510=1185.674,231.307,-62.316,-177.445,6.955,148.545
C00511=1185.669,231.556,-62.342,-177.443,6.957,148.545
C00512=1185.665,231.804,-62.368,-177.440,6.959,148.545
C00513=1185.661,232.053,-62.393,-177.438,6.961,148.545
C00514=1185.655,232.302,-62.419,-177.435,6.963,148.544
C00515=1185.651,232.550,-62.446,-177.432,6.966,148.544
C00516=1185.647,232.799,-62.471,-177.430,6.968,148.544
C00517=1185.643,233.047,-62.497,-177.428,6.970,148.544
C00518=1185.638,233.295,-62.523,-177.424,6.973,148.544
C00519=1185.634,233.544,-62.548,-177.422,6.975,148.544
C00520=1185.629,233.793,-62.575,-177.419,6.978,148.543
C00521=1185.624,234.042,-62.600,-177.417,6.980,148.543
C00522=1185.620,234.290,-62.626,-177.414,6.982,148.543
C00523=1185.615,234.539,-62.652,-177.411,6.985,148.543
C00524=1185.611,234.788,-62.679,-177.409,6.986,148.542
C00525=1185.606,235.036,-62.704,-177.406,6.989,148.542
C00526=1185.602,235.285,-62.730,-177.403,6.991,148.542
C00527=1185.597,235.533,-62.756,-177.401,6.993,148.542
C00528=1185.593,235.782,-62.781,-177.398,6.996,148.542
C00529=1185.589,236.031,-62.808,-177.396,6.998,148.542
C00530=1185.584,236.302,-62.836,-177.393,7.001,148.541
C00531=1185.579,236.573,-62.865,-177.389,7.003,148.541
C00532=1185.573,236.845,-62.893,-177.387,7.006,148.541
C00533=1185.569,237.117,-62.921,-177.384,7.008,148.541
C00534=1185.565,237.365,-62.948,-177.382,7.010,148.541
C00535=1185.561,237.614,-62.974,-177.379,7.013,148.540
C00536=1185.556,237.863,-63.000,-177.377,7.015,148.540
C00537=1185.551,238.111,-63.026,-177.373,7.018,148.540
C00538=1185.547,238.360,-63.052,-177.371,7.020,148.540
C00539=1185.542,238.609,-63.078,-177.368,7.023,148.539
C00540=1185.538,238.857,-63.105,-177.366,7.025,148.539
C00541=1185.534,239.106,-63.130,-177.363,7.027,148.539
C00542=1185.529,239.354,-63.158,-177.360,7.030,148.539
C00543=1185.524,239.602,-63.183,-177.358,7.031,148.539
C00544=1185.519,239.851,-63.209,-177.355,7.034,148.539
C00545=1185.515,240.100,-63.236,-177.353,7.037,148.538
C00546=1185.511,240.348,-63.261,-177.350,7.039,148.538
C00547=1185.507,240.597,-63.289,-177.347,7.041,148.538
C00548=1185.502,240.846,-63.314,-177.345,7.043,148.538
C00549=1185.498,241.094,-63.341,-177.342,7.046,148.538
C00550=1185.493,241.343,-63.367,-177.339,7.048,148.537
C00551=1185.489,241.591,-63.394,-177.337,7.051,148.537
C00552=1185.485,241.840,-63.420,-177.334,7.053,148.537
C00553=1185.480,242.088,-63.446,-177.331,7.056,148.537
C00554=1185.475,242.337,-63.472,-177.329,7.058,148.537
C00555=1185.471,242.585,-63.499,-177.326,7.061,148.537
C00556=1185.466,242.834,-63.525,-177.324,7.063,148.536
C00557=1185.462,243.082,-63.552,-177.321,7.064,148.536
C00558=1185.457,243.331,-63.578,-177.318,7.067,148.536
C00559=1185.453,243.580,-63.604,-177.316,7.070,148.536
C00560=1185.449,243.828,-63.631,-177.313,7.072,148.536
C00561=1185.444,244.077,-63.657,-177.311,7.074,148.536
C00562=1185.440,244.325,-63.684,-177.308,7.077,148.535
C00563=1185.436,244.574,-63.711,-177.305,7.079,148.535
C00564=1185.431,244.823,-63.737,-177.302,7.082,148.535
C00565=1185.426,245.071,-63.764,-177.300,7.084,148.535
C00566=1185.422,245.319,-63.791,-177.297,7.087,148.535
C00567=1185.417,245.569,-63.817,-177.295,7.089,148.534
C00568=1185.413,245.817,-63.843,-177.292,7.092,148.534
C00569=1185.409,246.065,-63.871,-177.290,7.094,148.534
C00570=1185.405,246.314,-63.896,-177.287,7.097,148.534
C00571=1185.400,246.563,-63.923,-177.284,7.099,148.534
C00572=1185.395,246.811,-63.950,-177.282,7.101,148.534
C00573=1185.391,247.059,-63.977,-177.279,7.104,148.534
C00574=1185.386,247.308,-64.003,-177.277,7.106,148.533
C00575=1185.382,247.557,-64.030,-177.274,7.108,148.533
C00576=1185.378,247.805,-64.057,-177.272,7.111,148.533
C00577=1185.373,248.054,-64.084,-177.269,7.114,148.533
C00578=1185.369,248.302,-64.110,-177.266,7.115,148.533
C00579=1185.364,248.551,-64.137,-177.263,7.118,148.533
C00580=1185.360,248.799,-64.164,-177.261,7.120,148.532
C00581=1185.355,249.048,-64.191,-177.258,7.123,148.532
C00582=1185.351,249.296,-64.217,-177.256,7.125,148.532
C00583=1185.346,249.544,-64.244,-177.253,7.128,148.532
C00584=1185.342,249.793,-64.271,-177.250,7.130,148.532
C00585=1185.338,250.042,-64.298,-177.248,7.133,148.532
C00586=1185.334,250.290,-64.325,-177.245,7.135,148.531
C00587=1185.329,250.539,-64.352,-177.242,7.138,148.531
C00588=1185.324,250.787,-64.379,-177.240,7.140,148.531
C00589=1185.321,251.036,-64.406,-177.237,7.143,148.531
C00590=1185.316,251.284,-64.433,-177.235,7.145,148.531
C00591=1185.311,251.533,-64.460,-177.232,7.148,148.531
C00592=1185.307,251.781,-64.487,-177.229,7.150,148.531
C00593=1185.303,252.029,-64.513,-177.227,7.153,148.530
C00594=1185.298,252.278,-64.541,-177.225,7.155,148.530
C00595=1185.294,252.527,-64.568,-177.221,7.157,148.530
C00596=1185.289,252.775,-64.595,-177.219,7.160,148.530
C00597=1185.285,253.024,-64.622,-177.216,7.163,148.530
C00598=1185.281,253.272,-64.649,-177.213,7.165,148.530
C00599=1185.276,253.521,-64.676,-177.211,7.167,148.530
C00600=1185.271,253.769,-64.703,-177.208,7.170,148.530
C00601=1185.267,254.018,-64.730,-177.206,7.173,148.529
C00602=1185.263,254.267,-64.757,-177.203,7.175,148.529
C00603=1185.258,254.515,-64.784,-177.201,7.177,148.529
C00604=1185.254,254.763,-64.811,-177.198,7.180,148.529
C00605=1185.250,255.011,-64.838,-177.195,7.182,148.529
C00606=1185.245,255.260,-64.865,-177.193,7.185,148.529
C00607=1185.240,255.508,-64.893,-177.191,7.187,148.529
C00608=1185.236,255.758,-64.920,-177.187,7.190,148.528
C00609=1185.232,256.006,-64.947,-177.185,7.192,148.528
C00610=1185.227,256.254,-64.975,-177.182,7.195,148.528
C00611=1185.223,256.502,-65.002,-177.180,7.198,148.528
C00612=1185.218,256.751,-65.029,-177.177,7.200,148.528
C00613=1185.214,257.000,-65.056,-177.174,7.203,148.528
C00614=1185.210,257.248,-65.084,-177.172,7.205,148.528
C00615=1185.206,257.496,-65.111,-177.169,7.208,148.528
C00616=1185.201,257.745,-65.138,-177.167,7.210,148.527
C00617=1185.197,257.994,-65.165,-177.164,7.213,148.527
C00618=1185.193,258.242,-65.193,-177.162,7.215,148.527
C00619=1185.188,258.490,-65.220,-177.159,7.218,148.527
C00620=1185.183,258.739,-65.247,-177.156,7.221,148.527
C00621=1185.180,258.987,-65.275,-177.154,7.223,148.527
C00622=1185.175,259.236,-65.302,-177.151,7.226,148.527
C00623=1185.171,259.484,-65.330,-177.149,7.228,148.526
C00624=1185.166,259.732,-65.357,-177.146,7.231,148.526
C00625=1185.162,259.981,-65.384,-177.144,7.233,148.526
C00626=1185.157,260.230,-65.413,-177.141,7.236,148.526
C00627=1185.152,260.478,-65.440,-177.138,7.239,148.526
C00628=1185.148,260.727,-65.468,-177.136,7.241,148.526
C00629=1185.144,260.975,-65.495,-177.133,7.244,148.526
C00630=1185.139,261.223,-65.523,-177.131,7.246,148.526
C00631=1185.135,261.471,-65.550,-177.128,7.249,148.526
C00632=1185.131,261.720,-65.578,-177.125,7.251,148.525
C00633=1185.126,261.969,-65.605,-177.123,7.253,148.525
C00634=1185.122,262.242,-65.636,-177.120,7.256,148.525
C00635=1185.116,262.514,-65.666,-177.117,7.259,148.525
C00636=1185.112,262.787,-65.696,-177.114,7.262,148.525
C00637=1185.107,263.060,-65.727,-177.111,7.265,148.525
C00638=1185.103,263.308,-65.754,-177.109,7.267,148.525
C00639=1185.098,263.558,-65.782,-177.106,7.270,148.524
C00640=1185.094,263.805,-65.810,-177.103,7.273,148.524
C00641=1185.089,264.054,-65.837,-177.101,7.275,148.524
C00642=1185.085,264.302,-65.865,-177.098,7.278,148.524
C00643=1185.081,264.550,-65.893,-177.095,7.281,148.524
C00644=1185.077,264.800,-65.921,-177.093,7.283,148.524
C00645=1185.072,265.048,-65.949,-177.090,7.286,148.524
C00646=1185.067,265.296,-65.977,-177.088,7.288,148.524
C00647=1185.063,265.545,-66.004,-177.085,7.291,148.524
C00648=1185.059,265.793,-66.032,-177.082,7.294,148.524
C00649=1185.054,266.041,-66.060,-177.080,7.296,148.523
C00650=1185.050,266.290,-66.088,-177.077,7.299,148.523
C00651=1185.046,266.538,-66.115,-177.075,7.301,148.523
C00652=1185.042,266.786,-66.144,-177.072,7.304,148.523
C00653=1185.037,267.035,-66.172,-177.069,7.307,148.523
C00654=1185.032,267.283,-66.199,-177.067,7.309,148.523
C00655=1185.028,267.532,-66.227,-177.064,7.312,148.523
C00656=1185.024,267.780,-66.255,-177.061,7.315,148.523
C00657=1185.019,268.029,-66.284,-177.059,7.317,148.523
C00658=1185.015,268.276,-66.311,-177.057,7.320,148.523
C00659=1185.011,268.526,-66.339,-177.054,7.322,148.523
C00660=1185.006,268.774,-66.367,-177.052,7.325,148.523
C00661=1185.002,269.022,-66.395,-177.048,7.328,148.522
C00662=1184.998,269.270,-66.423,-177.046,7.330,148.522
C00663=1184.993,269.518,-66.452,-177.044,7.333,148.522
C00664=1184.989,269.767,-66.480,-177.041,7.336,148.522
C00665=1184.984,270.015,-66.508,-177.039,7.338,148.522
C00666=1184.980,270.264,-66.536,-177.036,7.341,148.522
C00667=1184.976,270.512,-66.564,-177.033,7.344,148.522
C00668=1184.971,270.761,-66.593,-177.031,7.346,148.522
C00669=1184.967,271.009,-66.620,-177.028,7.349,148.522
C00670=1184.963,271.258,-66.648,-177.026,7.351,148.522
C00671=1184.958,271.506,-66.676,-177.023,7.354,148.521
C00672=1184.954,271.754,-66.704,-177.020,7.357,148.521
C00673=1184.949,272.003,-66.733,-177.018,7.359,148.521
C00674=1184.945,272.251,-66.761,-177.015,7.362,148.521
C00675=1184.940,272.499,-66.789,-177.012,7.365,148.521
C00676=1184.937,272.747,-66.818,-177.010,7.367,148.521
C00677=1184.932,272.995,-66.847,-177.007,7.370,148.521
C00678=1184.928,273.244,-66.875,-177.005,7.373,148.521
C00679=1184.924,273.493,-66.903,-177.002,7.375,148.521
C00680=1184.919,273.741,-66.931,-177.000,7.378,148.521
C00681=1184.915,273.989,-66.959,-176.997,7.381,148.521
C00682=1184.910,274.238,-66.988,-176.995,7.383,148.521
C00683=1184.906,274.486,-67.016,-176.992,7.386,148.521
C00684=1184.901,274.734,-67.044,-176.989,7.389,148.521
C00685=1184.897,274.983,-67.074,-176.987,7.391,148.520
C00686=1184.893,275.231,-67.102,-176.984,7.394,148.520
C00687=1184.888,275.479,-67.130,-176.981,7.397,148.520
C00688=1184.885,275.728,-67.158,-176.979,7.399,148.520
C00689=1184.880,275.976,-67.187,-176.976,7.402,148.520
C00690=1184.876,276.224,-67.216,-176.974,7.405,148.520
C00691=1184.872,276.473,-67.244,-176.971,7.408,148.520
C00692=1184.867,276.721,-67.272,-176.969,7.410,148.520
C00693=1184.863,276.970,-67.301,-176.966,7.413,148.520
C00694=1184.858,277.217,-67.330,-176.963,7.416,148.520
C00695=1184.854,277.466,-67.358,-176.961,7.418,148.520
C00696=1184.850,277.715,-67.387,-176.958,7.421,148.519
C00697=1184.845,277.963,-67.415,-176.955,7.424,148.519
C00698=1184.841,278.211,-67.444,-176.953,7.426,148.519
C00699=1184.837,278.460,-67.473,-176.950,7.429,148.519
C00700=1184.833,278.707,-67.501,-176.948,7.432,148.519
C00701=1184.828,278.956,-67.530,-176.945,7.434,148.519
C00702=1184.824,279.205,-67.559,-176.943,7.437,148.519
C00703=1184.820,279.452,-67.587,-176.940,7.440,148.519
C00704=1184.815,279.701,-67.616,-176.937,7.443,148.519
C00705=1184.811,279.950,-67.645,-176.935,7.446,148.519
C00706=1184.807,280.197,-67.673,-176.932,7.449,148.519
C00707=1184.802,280.446,-67.702,-176.930,7.452,148.519
C00708=1184.798,280.694,-67.731,-176.928,7.454,148.519
C00709=1184.793,280.942,-67.760,-176.925,7.457,148.519
C00710=1184.789,281.190,-67.789,-176.922,7.460,148.519
C00711=1184.785,281.439,-67.817,-176.919,7.463,148.519
C00712=1184.780,281.687,-67.846,-176.917,7.465,148.519
C00713=1184.776,281.936,-67.875,-176.914,7.468,148.519
C00714=1184.772,282.184,-67.904,-176.912,7.471,148.519
C00715=1184.768,282.433,-67.933,-176.910,7.473,148.519
C00716=1184.763,282.680,-67.962,-176.907,7.476,148.518
C00717=1184.758,282.929,-67.991,-176.904,7.479,148.518
C00718=1184.754,283.177,-68.020,-176.901,7.482,148.518
C00719=1184.751,283.425,-68.049,-176.899,7.484,148.518
C00720=1184.746,283.673,-68.077,-176.897,7.487,148.518
C00721=1184.742,283.922,-68.107,-176.894,7.490,148.518
C00722=1184.737,284.171,-68.135,-176.892,7.492,148.518
C00723=1184.733,284.419,-68.165,-176.889,7.495,148.518
C00724=1184.728,284.666,-68.194,-176.886,7.498,148.518
C00725=1184.724,284.915,-68.222,-176.883,7.501,148.518
C00726=1184.720,285.163,-68.252,-176.881,7.503,148.518
C00727=1184.716,285.412,-68.281,-176.879,7.506,148.518
C00728=1184.711,285.659,-68.310,-176.876,7.509,148.518
C00729=1184.707,285.908,-68.339,-176.873,7.512,148.518
C00730=1184.703,286.156,-68.368,-176.871,7.515,148.518
C00731=1184.698,286.405,-68.398,-176.868,7.518,148.518
C00732=1184.694,286.653,-68.427,-176.866,7.521,148.518
C00733=1184.689,286.901,-68.456,-176.863,7.524,148.518
C00734=1184.685,287.149,-68.485,-176.861,7.526,148.518
C00735=1184.681,287.397,-68.514,-176.858,7.529,148.518
C00736=1184.677,287.645,-68.543,-176.855,7.532,148.518
C00737=1184.673,287.894,-68.572,-176.853,7.535,148.518
C00738=1184.668,288.168,-68.605,-176.850,7.538,148.518
C00739=1184.663,288.443,-68.637,-176.847,7.541,148.518
C00740=1184.658,288.718,-68.670,-176.844,7.544,148.518
C00741=1184.654,288.993,-68.702,-176.841,7.546,148.517
C00742=1184.650,289.241,-68.732,-176.838,7.549,148.517
C00743=1184.645,289.488,-68.761,-176.836,7.553,148.517
C00744=1184.641,289.737,-68.790,-176.833,7.556,148.517
C00745=1184.637,289.985,-68.820,-176.831,7.558,148.517
C00746=1184.632,290.233,-68.849,-176.829,7.561,148.517
C00747=1184.628,290.482,-68.879,-176.826,7.564,148.517
C00748=1184.623,290.730,-68.908,-176.823,7.567,148.517
C00749=1184.619,290.978,-68.938,-176.821,7.569,148.517
C00750=1184.615,291.227,-68.967,-176.818,7.572,148.517
C00751=1184.611,291.475,-68.997,-176.816,7.575,148.517
C00752=1184.606,291.722,-69.026,-176.813,7.578,148.517
C00753=1184.602,291.971,-69.055,-176.811,7.580,148.517
C00754=1184.598,292.219,-69.085,-176.808,7.583,148.517
C00755=1184.593,292.467,-69.114,-176.805,7.586,148.517
C00756=1184.589,292.716,-69.144,-176.803,7.589,148.517
C00757=1184.585,292.964,-69.173,-176.800,7.592,148.517
C00758=1184.580,293.212,-69.203,-176.798,7.595,148.517
C00759=1184.576,293.461,-69.233,-176.795,7.598,148.517
C00760=1184.572,293.709,-69.262,-176.793,7.601,148.517
C00761=1184.568,293.957,-69.292,-176.790,7.604,148.517
C00762=1184.564,294.205,-69.322,-176.788,7.606,148.517
C00763=1184.560,294.453,-69.351,-176.785,7.609,148.517
C00764=1184.555,294.701,-69.381,-176.782,7.612,148.517
C00765=1184.550,294.950,-69.411,-176.780,7.615,148.517
C00766=1184.546,295.198,-69.440,-176.777,7.618,148.517
C00767=1184.542,295.446,-69.470,-176.775,7.620,148.517
C00768=1184.538,295.694,-69.500,-176.772,7.623,148.517
C00769=1184.534,295.942,-69.529,-176.770,7.626,148.517
C00770=1184.529,296.191,-69.559,-176.767,7.629,148.517
C00771=1184.525,296.439,-69.589,-176.764,7.632,148.517
C00772=1184.521,296.687,-69.619,-176.762,7.634,148.517
C00773=1184.517,296.935,-69.648,-176.759,7.637,148.517
C00774=1184.512,297.184,-69.678,-176.757,7.640,148.517
C00775=1184.508,297.431,-69.709,-176.754,7.643,148.517
C00776=1184.504,297.680,-69.738,-176.751,7.646,148.517
C00777=1184.499,297.928,-69.768,-176.750,7.649,148.517
C00778=1184.495,298.176,-69.798,-176.747,7.652,148.517
C00779=1184.491,298.424,-69.828,-176.744,7.655,148.517
C00780=1184.487,298.672,-69.857,-176.741,7.658,148.517
C00781=1184.482,298.920,-69.888,-176.739,7.661,148.517
C00782=1184.478,299.169,-69.917,-176.737,7.663,148.517
C00783=1184.474,299.416,-69.948,-176.734,7.666,148.517
C00784=1184.469,299.665,-69.978,-176.732,7.669,148.517
C00785=1184.466,299.913,-70.008,-176.729,7.672,148.517
C00786=1184.461,300.162,-70.038,-176.726,7.675,148.517
C00787=1184.457,300.409,-70.068,-176.723,7.678,148.517
C00788=1184.453,300.658,-70.098,-176.721,7.680,148.517
C00789=1184.448,300.906,-70.129,-176.719,7.683,148.517
C00790=1184.444,301.154,-70.158,-176.716,7.687,148.517
C00791=1184.440,301.402,-70.189,-176.714,7.690,148.517
C00792=1184.435,301.650,-70.218,-176.711,7.693,148.517
C00793=1184.431,301.898,-70.248,-176.708,7.696,148.517
C00794=1184.427,302.146,-70.278,-176.706,7.698,148.517
C00795=1184.423,302.395,-70.309,-176.703,7.701,148.517
C00796=1184.418,302.643,-70.339,-176.701,7.704,148.517
C00797=1184.414,302.891,-70.369,-176.698,7.707,148.517
C00798=1184.410,303.139,-70.400,-176.696,7.710,148.517
C00799=1184.406,303.387,-70.429,-176.693,7.712,148.517
C00800=1184.401,303.635,-70.460,-176.691,7.715,148.517
C00801=1184.397,303.883,-70.490,-176.689,7.719,148.517
C00802=1184.393,304.132,-70.521,-176.686,7.722,148.517
C00803=1184.389,304.380,-70.551,-176.683,7.725,148.517
C00804=1184.384,304.628,-70.582,-176.680,7.728,148.517
C00805=1184.380,304.876,-70.611,-176.678,7.731,148.517
C00806=1184.376,305.124,-70.642,-176.676,7.733,148.517
C00807=1184.372,305.372,-70.672,-176.673,7.736,148.517
C00808=1184.367,305.621,-70.702,-176.671,7.739,148.517
C00809=1184.363,305.869,-70.733,-176.668,7.742,148.517
C00810=1184.359,306.116,-70.763,-176.666,7.745,148.517
C00811=1184.354,306.364,-70.794,-176.663,7.748,148.517
C00812=1184.350,306.612,-70.824,-176.661,7.751,148.517
C00813=1184.346,306.861,-70.855,-176.658,7.754,148.517
C00814=1184.342,307.109,-70.885,-176.656,7.757,148.517
C00815=1184.338,307.357,-70.916,-176.653,7.760,148.517
C00816=1184.333,307.605,-70.946,-176.650,7.763,148.517
C00817=1184.329,307.852,-70.977,-176.648,7.766,148.517
C00818=1184.325,308.101,-71.008,-176.645,7.769,148.517
C00819=1184.320,308.350,-71.038,-176.643,7.771,148.517
C00820=1184.316,308.597,-71.068,-176.640,7.774,148.517
C00821=1184.312,308.845,-71.099,-176.638,7.777,148.517
C00822=1184.308,309.094,-71.130,-176.635,7.781,148.518
C00823=1184.304,309.342,-71.160,-176.633,7.784,148.518
C00824=1184.299,309.590,-71.191,-176.630,7.787,148.517
C00825=1184.295,309.838,-71.222,-176.627,7.790,148.517
C00826=1184.291,310.086,-71.252,-176.626,7.792,148.518
C00827=1184.287,310.334,-71.283,-176.623,7.795,148.518
C00828=1184.282,310.582,-71.314,-176.620,7.798,148.518
C00829=1184.278,310.830,-71.345,-176.617,7.801,148.518
C00830=1184.274,311.078,-71.375,-176.615,7.805,148.518
C00831=1184.270,311.326,-71.406,-176.612,7.808,148.518
C00832=1184.266,311.575,-71.437,-176.610,7.811,148.518
C00833=1184.261,311.823,-71.468,-176.608,7.813,148.518
C00834=1184.257,312.070,-71.498,-176.605,7.816,148.518
C00835=1184.253,312.319,-71.529,-176.603,7.819,148.518
C00836=1184.249,312.566,-71.560,-176.600,7.822,148.518
C00837=1184.244,312.814,-71.591,-176.598,7.825,148.518
C00838=1184.241,313.063,-71.622,-176.595,7.828,148.518
C00839=1184.236,313.311,-71.652,-176.593,7.832,148.518
C00840=1184.232,313.559,-71.683,-176.590,7.835,148.518
C00841=1184.228,313.807,-71.714,-176.588,7.837,148.518
C00842=1184.223,314.083,-71.749,-176.585,7.841,148.518
C00843=1184.218,314.360,-71.784,-176.582,7.844,148.518
C00844=1184.213,314.637,-71.818,-176.580,7.847,148.518
C00845=1184.209,314.913,-71.852,-176.576,7.851,148.518
C00846=1184.205,315.161,-71.883,-176.574,7.854,148.519
C00847=1184.200,315.409,-71.915,-176.571,7.857,148.519
C00848=1184.196,315.657,-71.946,-176.569,7.859,148.519
C00849=1184.192,315.905,-71.977,-176.567,7.863,148.519
C00850=1184.188,316.154,-72.008,-176.564,7.866,148.519
C00851=1184.183,316.401,-72.039,-176.562,7.869,148.519
C00852=1184.179,316.649,-72.070,-176.559,7.872,148.519
C00853=1184.176,316.898,-72.100,-176.557,7.875,148.519
C00854=1184.171,317.145,-72.132,-176.554,7.878,148.519
C00855=1184.167,317.394,-72.163,-176.552,7.881,148.519
C00856=1184.163,317.642,-72.194,-176.549,7.884,148.519
C00857=1184.159,317.890,-72.226,-176.547,7.887,148.519
C00858=1184.154,318.138,-72.256,-176.544,7.890,148.519
C00859=1184.150,318.385,-72.288,-176.542,7.893,148.519
C00860=1184.146,318.634,-72.319,-176.539,7.896,148.519
C00861=1184.142,318.881,-72.351,-176.537,7.899,148.519
C00862=1184.138,319.130,-72.382,-176.535,7.902,148.520
C00863=1184.133,319.378,-72.412,-176.532,7.905,148.520
C00864=1184.129,319.626,-72.444,-176.529,7.908,148.520
C00865=1184.125,319.874,-72.475,-176.527,7.912,148.520
C00866=1184.121,320.122,-72.507,-176.524,7.915,148.520
C00867=1184.116,320.370,-72.538,-176.522,7.917,148.520
C00868=1184.113,320.618,-72.570,-176.520,7.920,148.520
C00869=1184.108,320.865,-72.601,-176.517,7.924,148.520
C00870=1184.104,321.114,-72.632,-176.515,7.927,148.520
C00871=1184.099,321.361,-72.664,-176.512,7.930,148.520
C00872=1184.095,321.610,-72.695,-176.510,7.933,148.520
C00873=1184.091,321.857,-72.727,-176.507,7.936,148.520
C00874=1184.087,322.106,-72.758,-176.505,7.939,148.521
C00875=1184.083,322.353,-72.789,-176.502,7.942,148.521
C00876=1184.079,322.601,-72.821,-176.500,7.945,148.521
C00877=1184.075,322.850,-72.852,-176.497,7.948,148.521
C00878=1184.071,323.097,-72.884,-176.495,7.951,148.521
C00879=1184.067,323.345,-72.916,-176.493,7.954,148.521
C00880=1184.062,323.594,-72.947,-176.490,7.957,148.521
C00881=1184.058,323.842,-72.979,-176.488,7.960,148.521
C00882=1184.054,324.089,-73.010,-176.486,7.964,148.521
C00883=1184.050,324.337,-73.042,-176.483,7.967,148.521
C00884=1184.046,324.586,-73.073,-176.481,7.970,148.522
C00885=1184.042,324.833,-73.105,-176.478,7.973,148.522
C00886=1184.037,325.081,-73.137,-176.476,7.976,148.522
C00887=1184.033,325.329,-73.169,-176.473,7.979,148.522
C00888=1184.029,325.577,-73.200,-176.471,7.983,148.522
C00889=1184.025,325.825,-73.232,-176.468,7.986,148.522
C00890=1184.021,326.073,-73.263,-176.466,7.988,148.522
C00891=1184.016,326.321,-73.296,-176.463,7.991,148.522
C00892=1184.012,326.568,-73.327,-176.461,7.994,148.522
C00893=1184.008,326.816,-73.359,-176.459,7.997,148.522
C00894=1184.005,327.064,-73.391,-176.456,8.001,148.522
C00895=1183.999,327.313,-73.422,-176.454,8.004,148.522
C00896=1183.996,327.561,-73.454,-176.451,8.007,148.523
C00897=1183.992,327.809,-73.486,-176.449,8.010,148.523
C00898=1183.987,328.056,-73.518,-176.446,8.013,148.523
C00899=1183.983,328.305,-73.550,-176.444,8.017,148.523
C00900=1183.979,328.552,-73.581,-176.441,8.020,148.523
C00901=1183.974,328.800,-73.614,-176.439,8.023,148.523
C00902=1183.971,329.048,-73.646,-176.436,8.026,148.523
C00903=1183.966,329.296,-73.677,-176.434,8.029,148.524
C00904=1183.962,329.544,-73.709,-176.432,8.032,148.524
C00905=1183.958,329.792,-73.741,-176.430,8.035,148.524
C00906=1183.954,330.039,-73.773,-176.427,8.038,148.524
C00907=1183.949,330.288,-73.805,-176.425,8.041,148.524
C00908=1183.946,330.536,-73.837,-176.423,8.044,148.524
C00909=1183.942,330.784,-73.869,-176.420,8.048,148.524
C00910=1183.937,331.031,-73.901,-176.418,8.051,148.524
C00911=1183.933,331.279,-73.933,-176.415,8.054,148.525
C00912=1183.929,331.528,-73.965,-176.413,8.057,148.525
C00913=1183.925,331.774,-73.997,-176.410,8.060,148.525
C00914=1183.920,332.023,-74.030,-176.408,8.064,148.525
C00915=1183.917,332.271,-74.062,-176.405,8.067,148.525
C00916=1183.913,332.519,-74.094,-176.403,8.070,148.525
C00917=1183.908,332.767,-74.126,-176.401,8.073,148.525
C00918=1183.904,333.015,-74.158,-176.398,8.076,148.525
C00919=1183.900,333.262,-74.191,-176.396,8.080,148.526
C00920=1183.896,333.510,-74.223,-176.394,8.083,148.526
C00921=1183.891,333.758,-74.255,-176.391,8.086,148.526
C00922=1183.888,334.006,-74.286,-176.389,8.088,148.526
C00923=1183.883,334.254,-74.319,-176.387,8.092,148.526
C00924=1183.880,334.502,-74.351,-176.384,8.095,148.526
C00925=1183.875,334.749,-74.384,-176.382,8.098,148.526
C00926=1183.871,334.998,-74.415,-176.380,8.101,148.527
C00927=1183.867,335.245,-74.449,-176.377,8.105,148.527
C00928=1183.863,335.493,-74.480,-176.375,8.108,148.527
C00929=1183.859,335.742,-74.513,-176.373,8.111,148.527
C00930=1183.854,335.989,-74.546,-176.370,8.114,148.527
C00931=1183.850,336.237,-74.577,-176.368,8.117,148.527
C00932=1183.846,336.485,-74.610,-176.365,8.121,148.527
C00933=1183.842,336.732,-74.642,-176.363,8.124,148.528
C00934=1183.838,336.981,-74.675,-176.361,8.127,148.528
C00935=1183.834,337.229,-74.707,-176.359,8.131,148.528
C00936=1183.830,337.476,-74.740,-176.356,8.134,148.528
C00937=1183.825,337.724,-74.772,-176.354,8.137,148.528
C00938=1183.822,337.972,-74.805,-176.351,8.140,148.529
C00939=1183.817,338.220,-74.837,-176.349,8.144,148.529
C00940=1183.813,338.468,-74.870,-176.346,8.147,148.529
C00941=1183.809,338.716,-74.902,-176.344,8.150,148.529
C00942=1183.805,338.963,-74.935,-176.342,8.153,148.529
C00943=1183.800,339.211,-74.967,-176.340,8.157,148.529
C00944=1183.797,339.459,-75.000,-176.337,8.160,148.530
C00945=1183.792,339.707,-75.032,-176.335,8.163,148.530
C00946=1183.788,339.985,-75.069,-176.332,8.166,148.530
C00947=1183.783,340.265,-75.106,-176.330,8.170,148.530
C00948=1183.779,340.544,-75.143,-176.327,8.174,148.530
C00949=1183.774,340.822,-75.179,-176.325,8.177,148.531
C00950=1183.770,341.071,-75.212,-176.323,8.180,148.531
C00951=1183.766,341.318,-75.245,-176.320,8.183,148.531
C00952=1183.761,341.567,-75.277,-176.318,8.187,148.531
C00953=1183.758,341.814,-75.310,-176.316,8.190,148.531
C00954=1183.753,342.061,-75.343,-176.313,8.193,148.531
C00955=1183.749,342.309,-75.375,-176.311,8.197,148.532
C00956=1183.745,342.557,-75.408,-176.309,8.200,148.532
C00957=1183.741,342.805,-75.442,-176.306,8.203,148.532
C00958=1183.737,343.052,-75.474,-176.304,8.206,148.532
C00959=1183.733,343.301,-75.507,-176.302,8.210,148.532
C00960=1183.729,343.548,-75.540,-176.300,8.213,148.533
C00961=1183.724,343.796,-75.573,-176.297,8.216,148.533
C00962=1183.720,344.044,-75.605,-176.295,8.219,148.533
C00963=1183.716,344.292,-75.638,-176.292,8.223,148.533
C00964=1183.712,344.540,-75.671,-176.290,8.226,148.533
C00965=1183.708,344.787,-75.704,-176.288,8.229,148.534
C00966=1183.704,345.035,-75.737,-176.286,8.233,148.534
C00967=1183.700,345.283,-75.770,-176.283,8.236,148.534
C00968=1183.696,345.531,-75.803,-176.281,8.239,148.534
C00969=1183.691,345.779,-75.836,-176.279,8.243,148.534
C00970=1183.687,346.027,-75.869,-176.277,8.246,148.535
C00971=1183.683,346.274,-75.902,-176.274,8.249,148.535
C00972=1183.679,346.522,-75.936,-176.272,8.253,148.535
C00973=1183.676,346.769,-75.968,-176.270,8.256,148.535
C00974=1183.671,347.017,-76.001,-176.268,8.259,148.536
C00975=1183.667,347.265,-76.034,-176.265,8.263,148.536
C00976=1183.663,347.513,-76.067,-176.263,8.266,148.536
C00977=1183.659,347.761,-76.100,-176.261,8.269,148.536
C00978=1183.655,348.009,-76.133,-176.259,8.273,148.537
C00979=1183.650,348.256,-76.166,-176.257,8.276,148.537
C00980=1183.646,348.504,-76.200,-176.255,8.279,148.537
C00981=1183.642,348.752,-76.233,-176.252,8.283,148.537
C00982=1183.638,349.000,-76.266,-176.250,8.286,148.537
C00983=1183.634,349.247,-76.299,-176.248,8.289,148.538
C00984=1183.630,349.495,-76.332,-176.246,8.293,148.538
C00985=1183.626,349.742,-76.366,-176.243,8.296,148.538
C00986=1183.622,349.990,-76.399,-176.241,8.299,148.538
C00987=1183.618,350.238,-76.432,-176.239,8.303,148.539
C00988=1183.614,350.486,-76.466,-176.237,8.306,148.539
C00989=1183.610,350.734,-76.499,-176.235,8.310,148.539
C00990=1183.606,350.982,-76.532,-176.232,8.313,148.539
C00991=1183.601,351.230,-76.566,-176.230,8.316,148.540
C00992=1183.597,351.477,-76.599,-176.228,8.320,148.540
C00993=1183.593,351.725,-76.632,-176.226,8.323,148.540
C00994=1183.589,351.972,-76.666,-176.224,8.326,148.541
C00995=1183.585,352.220,-76.699,-176.222,8.330,148.541
C00996=1183.581,352.468,-76.732,-176.219,8.333,148.541
C00997=1183.577,352.716,-76.766,-176.217,8.336,148.541
C00998=1183.573,352.964,-76.799,-176.215,8.340,148.542
C00999=1183.569,353.211,-76.833,-176.213,8.343,148.542
C01000=1183.565,353.459,-76.866,-176.211,8.347,148.542
C01001=1183.560,353.707,-76.900,-176.208,8.350,148.542
C01002=1183.556,353.954,-76.934,-176.207,8.354,148.543
C01003=1183.552,354.201,-76.967,-176.204,8.357,148.543
C01004=1183.549,354.450,-77.000,-176.202,8.360,148.543
C01005=1183.544,354.698,-77.034,-176.200,8.364,148.544
C01006=1183.541,354.945,-77.067,-176.198,8.367,148.544
C01007=1183.536,355.193,-77.101,-176.196,8.371,148.544
C01008=1183.532,355.441,-77.134,-176.194,8.374,148.544
C01009=1183.528,355.688,-77.168,-176.192,8.377,148.545
C01010=1183.524,355.936,-77.202,-176.190,8.381,148.545
C01011=1183.520,356.183,-77.236,-176.188,8.384,148.545
C01012=1183.516,356.431,-77.269,-176.185,8.388,148.546
C01013=1183.511,356.679,-77.303,-176.183,8.391,148.546
C01014=1183.508,356.927,-77.337,-176.181,8.395,148.546
C01015=1183.504,357.174,-77.370,-176.179,8.398,148.546
C01016=1183.499,357.422,-77.404,-176.177,8.401,148.547
C01017=1183.495,357.670,-77.438,-176.175,8.405,148.547
C01018=1183.491,357.917,-77.471,-176.173,8.408,148.547
C01019=1183.487,358.166,-77.506,-176.171,8.412,148.548
C01020=1183.483,358.413,-77.539,-176.169,8.415,148.548
C01021=1183.479,358.660,-77.573,-176.167,8.419,148.548
C01022=1183.475,358.907,-77.606,-176.165,8.422,148.549
C01023=1183.471,359.156,-77.641,-176.163,8.426,148.549
C01024=1183.467,359.403,-77.674,-176.161,8.429,148.549
C01025=1183.463,359.651,-77.708,-176.159,8.433,148.550
C01026=1183.459,359.899,-77.742,-176.157,8.436,148.550
C01027=1183.455,360.146,-77.776,-176.155,8.440,148.550
C01028=1183.451,360.394,-77.809,-176.152,8.443,148.551
C01029=1183.447,360.641,-77.844,-176.151,8.447,148.551
C01030=1183.443,360.889,-77.878,-176.149,8.450,148.551
C01031=1183.439,361.137,-77.912,-176.147,8.453,148.552
C01032=1183.435,361.384,-77.946,-176.145,8.457,148.552
C01033=1183.431,361.632,-77.980,-176.143,8.461,148.553
C01034=1183.427,361.880,-78.014,-176.141,8.464,148.553
C01035=1183.423,362.127,-78.048,-176.139,8.468,148.553
C01036=1183.420,362.375,-78.082,-176.137,8.471,148.554
C01037=1183.415,362.623,-78.116,-176.135,8.475,148.554
C01038=1183.411,362.870,-78.149,-176.133,8.478,148.554
C01039=1183.407,363.118,-78.184,-176.131,8.482,148.555
C01040=1183.403,363.366,-78.218,-176.129,8.485,148.555
C01041=1183.398,363.614,-78.252,-176.127,8.489,148.555
C01042=1183.395,363.861,-78.286,-176.126,8.492,148.556
C01043=1183.390,364.109,-78.321,-176.124,8.495,148.556
C01044=1183.387,364.356,-78.354,-176.122,8.499,148.557
C01045=1183.383,364.604,-78.389,-176.120,8.502,148.557
C01046=1183.378,364.852,-78.422,-176.119,8.506,148.557
C01047=1183.375,365.099,-78.456,-176.116,8.509,148.558
C01048=1183.371,365.347,-78.491,-176.114,8.513,148.558
C01049=1183.367,365.594,-78.525,-176.113,8.517,148.559
C01050=1183.362,365.876,-78.565,-176.111,8.520,148.559
C01051=1183.358,366.157,-78.603,-176.109,8.524,148.559
C01052=1183.353,366.439,-78.642,-176.107,8.529,148.560
C01053=1183.348,366.721,-78.681,-176.105,8.532,148.561
C01054=1183.344,366.968,-78.715,-176.103,8.536,148.561
C01055=1183.341,367.216,-78.750,-176.102,8.539,148.561
C01056=1183.336,367.463,-78.784,-176.100,8.542,148.562
C01057=1183.332,367.710,-78.818,-176.099,8.546,148.562
C01058=1183.328,367.958,-78.853,-176.097,8.550,148.563
C01059=1183.324,368.206,-78.887,-176.095,8.553,148.563
C01060=1183.320,368.454,-78.922,-176.093,8.557,148.564
C01061=1183.316,368.701,-78.956,-176.092,8.560,148.564
C01062=1183.312,368.948,-78.990,-176.090,8.563,148.564
C01063=1183.308,369.196,-79.025,-176.089,8.567,148.565
C01064=1183.304,369.444,-79.059,-176.087,8.571,148.565
C01065=1183.300,369.692,-79.093,-176.086,8.574,148.566
C01066=1183.296,369.939,-79.128,-176.084,8.577,148.566
C01067=1183.292,370.187,-79.163,-176.082,8.581,148.567
C01068=1183.288,370.434,-79.197,-176.081,8.584,148.567
C01069=1183.284,370.682,-79.231,-176.079,8.587,148.568
C01070=1183.280,370.929,-79.267,-176.078,8.591,148.568
C01071=1183.276,371.177,-79.301,-176.077,8.594,148.569
C01072=1183.272,371.424,-79.335,-176.075,8.598,148.569
C01073=1183.267,371.672,-79.370,-176.073,8.601,148.570
C01074=1183.264,371.920,-79.404,-176.072,8.605,148.570
C01075=1183.260,372.167,-79.438,-176.071,8.608,148.571
C01076=1183.256,372.415,-79.473,-176.069,8.612,148.571
C01077=1183.252,372.662,-79.508,-176.068,8.615,148.572
C01078=1183.248,372.910,-79.543,-176.066,8.618,148.572
C01079=1183.243,373.157,-79.577,-176.065,8.622,148.573
C01080=1183.240,373.405,-79.612,-176.063,8.625,148.573
C01081=1183.236,373.652,-79.647,-176.062,8.629,148.574
C01082=1183.232,373.900,-79.681,-176.061,8.632,148.574
C01083=1183.228,374.148,-79.716,-176.059,8.636,148.575
C01084=1183.223,374.395,-79.751,-176.058,8.639,148.575
C01085=1183.221,374.643,-79.786,-176.057,8.643,148.576
C01086=1183.216,374.890,-79.820,-176.056,8.645,148.576
C01087=1183.212,375.138,-79.855,-176.054,8.649,148.577
C01088=1183.207,375.386,-79.889,-176.053,8.652,148.577
C01089=1183.205,375.633,-79.924,-176.052,8.656,148.578
C01090=1183.200,375.880,-79.959,-176.051,8.659,148.578
C01091=1183.196,376.128,-79.994,-176.049,8.663,148.579
C01092=1183.192,376.375,-80.029,-176.048,8.666,148.579
C01093=1183.188,376.623,-80.064,-176.047,8.670,148.580
C01094=1183.183,376.871,-80.098,-176.045,8.673,148.580
C01095=1183.180,377.118,-80.133,-176.045,8.676,148.581
C01096=1183.176,377.366,-80.168,-176.043,8.680,148.582
C01097=1183.172,377.613,-80.203,-176.042,8.682,148.582
C01098=1183.168,377.861,-80.238,-176.041,8.686,148.583
C01099=1183.163,378.108,-80.272,-176.040,8.689,148.583
C01100=1183.160,378.356,-80.308,-176.039,8.692,148.584
C01101=1183.156,378.603,-80.342,-176.037,8.696,148.584
C01102=1183.152,378.850,-80.377,-176.036,8.699,148.585
C01103=1183.148,379.099,-80.412,-176.036,8.702,148.585
C01104=1183.144,379.345,-80.447,-176.034,8.706,148.586
C01105=1183.140,379.593,-80.482,-176.033,8.709,148.587
C01106=1183.136,379.841,-80.517,-176.033,8.712,148.587
C01107=1183.132,380.088,-80.552,-176.032,8.715,148.588
C01108=1183.128,380.337,-80.587,-176.030,8.719,148.588
C01109=1183.124,380.583,-80.622,-176.029,8.722,148.589
C01110=1183.120,380.831,-80.657,-176.028,8.725,148.589
C01111=1183.116,381.078,-80.692,-176.027,8.728,148.590
C01112=1183.112,381.326,-80.727,-176.027,8.731,148.591
C01113=1183.109,381.574,-80.762,-176.026,8.735,148.591
C01114=1183.104,381.820,-80.797,-176.024,8.738,148.592
C01115=1183.100,382.068,-80.832,-176.024,8.742,148.592
C01116=1183.097,382.316,-80.868,-176.023,8.745,148.593
C01117=1183.092,382.563,-80.902,-176.022,8.748,148.594
C01118=1183.088,382.811,-80.938,-176.021,8.751,148.594
C01119=1183.084,383.058,-80.972,-176.020,8.754,148.595
C01120=1183.080,383.306,-81.008,-176.020,8.757,148.595
C01121=1183.077,383.553,-81.043,-176.019,8.760,148.596
C01122=1183.072,383.801,-81.078,-176.018,8.764,148.597
C01123=1183.068,384.048,-81.113,-176.018,8.767,148.597
C01124=1183.064,384.296,-81.148,-176.017,8.770,148.598
C01125=1183.060,384.543,-81.183,-176.016,8.773,148.598
C01126=1183.056,384.791,-81.219,-176.015,8.776,148.599
C01127=1183.052,385.039,-81.254,-176.014,8.779,148.600
C01128=1183.048,385.286,-81.289,-176.013,8.782,148.600
C01129=1183.044,385.533,-81.324,-176.013,8.785,148.601
C01130=1183.041,385.781,-81.359,-176.012,8.789,148.601
C01131=1183.036,386.028,-81.394,-176.012,8.791,148.602
C01132=1183.033,386.275,-81.430,-176.011,8.794,148.603
C01133=1183.029,386.524,-81.465,-176.010,8.797,148.603
C01134=1183.024,386.770,-81.500,-176.010,8.800,148.604
C01135=1183.021,387.018,-81.536,-176.009,8.804,148.605
C01136=1183.017,387.265,-81.571,-176.009,8.806,148.605
C01137=1183.012,387.513,-81.606,-176.009,8.809,148.606
C01138=1183.009,387.760,-81.641,-176.008,8.812,148.606
C01139=1183.005,388.008,-81.677,-176.007,8.815,148.607
C01140=1183.001,388.255,-81.712,-176.007,8.818,148.608
C01141=1182.997,388.503,-81.747,-176.006,8.821,148.608
C01142=1182.993,388.751,-81.783,-176.005,8.824,148.609
C01143=1182.989,388.998,-81.818,-176.005,8.826,148.609
C01144=1182.985,389.245,-81.853,-176.005,8.830,148.610
C01145=1182.981,389.493,-81.888,-176.004,8.833,148.611
C01146=1182.977,389.740,-81.924,-176.004,8.835,148.611
C01147=1182.973,389.988,-81.959,-176.003,8.839,148.612
C01148=1182.969,390.235,-81.995,-176.003,8.841,148.613
C01149=1182.965,390.482,-82.030,-176.003,8.844,148.613
C01150=1182.961,390.730,-82.065,-176.002,8.846,148.614
C01151=1182.957,390.977,-82.100,-176.002,8.850,148.615
C01152=1182.953,391.225,-82.136,-176.002,8.852,148.615
C01153=1182.949,391.473,-82.172,-176.001,8.855,148.616
C01154=1182.944,391.757,-82.212,-176.001,8.859,148.617
C01155=1182.940,392.040,-82.253,-176.001,8.861,148.617
C01156=1182.936,392.325,-82.293,-176.000,8.865,148.618
C01157=1182.931,392.608,-82.334,-176.000,8.868,148.619
C01158=1182.928,392.855,-82.369,-176.000,8.870,148.619
C01159=1182.923,393.103,-82.406,-175.999,8.873,148.620
C01160=1182.919,393.350,-82.441,-175.999,8.876,148.621
C01161=1182.915,393.598,-82.476,-175.998,8.879,148.621
C01162=1182.911,393.846,-82.511,-175.999,8.882,148.622
C01163=1182.908,394.093,-82.547,-175.998,8.884,148.623
C01164=1182.903,394.340,-82.582,-175.998,8.887,148.623
C01165=1182.900,394.588,-82.617,-175.998,8.889,148.624
C01166=1182.895,394.835,-82.654,-175.998,8.892,148.625
C01167=1182.892,395.083,-82.689,-175.998,8.894,148.625
C01168=1182.887,395.330,-82.724,-175.997,8.898,148.626
C01169=1182.884,395.577,-82.760,-175.997,8.900,148.626
C01170=1182.880,395.825,-82.795,-175.997,8.902,148.627
C01171=1182.876,396.072,-82.832,-175.997,8.905,148.628
C01172=1182.872,396.319,-82.867,-175.996,8.908,148.628
C01173=1182.868,396.567,-82.902,-175.996,8.910,148.629
C01174=1182.864,396.815,-82.937,-175.996,8.913,148.629
C01175=1182.860,397.062,-82.973,-175.996,8.915,148.630
C01176=1182.856,397.310,-83.009,-175.996,8.918,148.631
C01177=1182.852,397.557,-83.044,-175.996,8.920,148.631
C01178=1182.848,397.804,-83.080,-175.995,8.923,148.632
C01179=1182.844,398.052,-83.115,-175.995,8.926,148.633
C01180=1182.841,398.299,-83.151,-175.995,8.928,148.633
C01181=1182.836,398.547,-83.186,-175.995,8.931,148.634
C01182=1182.832,398.794,-83.222,-175.995,8.933,148.634
C01183=1182.828,399.042,-83.258,-175.995,8.935,148.635
C01184=1182.825,399.289,-83.293,-175.995,8.938,148.636
C01185=1182.820,399.537,-83.329,-175.995,8.940,148.636
C01186=1182.816,399.784,-83.364,-175.995,8.943,148.637
C01187=1182.812,400.031,-83.400,-175.995,8.945,148.638
C01188=1182.809,400.279,-83.435,-175.995,8.947,148.638
C01189=1182.805,400.526,-83.471,-175.995,8.950,148.639
C01190=1182.801,400.774,-83.507,-175.995,8.952,148.639
C01191=1182.796,401.021,-83.542,-175.994,8.955,148.640
C01192=1182.793,401.268,-83.578,-175.995,8.957,148.641
C01193=1182.789,401.516,-83.613,-175.994,8.959,148.641
C01194=1182.785,401.763,-83.650,-175.995,8.962,148.642
C01195=1182.781,402.011,-83.686,-175.994,8.964,148.642
C01196=1182.777,402.257,-83.721,-175.994,8.967,148.643
C01197=1182.773,402.505,-83.757,-175.994,8.969,148.644
C01198=1182.769,402.753,-83.793,-175.994,8.971,148.644
C01199=1182.765,403.000,-83.828,-175.994,8.974,148.645
C01200=1182.762,403.248,-83.864,-175.994,8.975,148.645
C01201=1182.757,403.495,-83.900,-175.995,8.978,148.646
C01202=1182.753,403.742,-83.935,-175.994,8.980,148.647
C01203=1182.749,403.990,-83.971,-175.994,8.983,148.647
C01204=1182.746,404.237,-84.006,-175.994,8.985,148.648
C01205=1182.741,404.485,-84.042,-175.994,8.987,148.648
C01206=1182.737,404.733,-84.078,-175.994,8.990,148.649
C01207=1182.734,404.979,-84.114,-175.994,8.991,148.650
C01208=1182.729,405.227,-84.150,-175.994,8.993,148.650
C01209=1182.725,405.474,-84.186,-175.994,8.996,148.651
C01210=1182.722,405.722,-84.221,-175.994,8.998,148.651
C01211=1182.718,405.969,-84.257,-175.994,9.001,148.652
C01212=1182.714,406.217,-84.293,-175.995,9.002,148.653
C01213=1182.709,406.464,-84.328,-175.994,9.005,148.653
C01214=1182.706,406.711,-84.363,-175.994,9.007,148.654
C01215=1182.702,406.958,-84.400,-175.994,9.009,148.654
C01216=1182.698,407.206,-84.436,-175.995,9.011,148.655
C01217=1182.694,407.453,-84.471,-175.995,9.013,148.655
C01218=1182.690,407.701,-84.508,-175.994,9.016,148.656
C01219=1182.686,407.948,-84.543,-175.994,9.018,148.656
C01220=1182.682,408.195,-84.578,-175.995,9.020,148.657
C01221=1182.679,408.442,-84.615,-175.995,9.022,148.658
C01222=1182.674,408.690,-84.651,-175.994,9.024,148.658
C01223=1182.671,408.938,-84.686,-175.995,9.026,148.659
C01224=1182.667,409.185,-84.722,-175.995,9.028,148.659
C01225=1182.663,409.433,-84.758,-175.995,9.030,148.660
C01226=1182.658,409.680,-84.793,-175.995,9.032,148.660
C01227=1182.655,409.927,-84.829,-175.995,9.034,148.661
C01228=1182.651,410.174,-84.866,-175.995,9.037,148.662
C01229=1182.647,410.422,-84.901,-175.995,9.038,148.662
C01230=1182.643,410.669,-84.937,-175.995,9.041,148.663
C01231=1182.639,410.917,-84.973,-175.995,9.043,148.663
C01232=1182.635,411.164,-85.009,-175.995,9.044,148.664
C01233=1182.631,411.411,-85.044,-175.995,9.047,148.664
C01234=1182.627,411.659,-85.080,-175.995,9.049,148.665
C01235=1182.623,411.906,-85.116,-175.996,9.051,148.665
C01236=1182.619,412.154,-85.152,-175.995,9.053,148.666
C01237=1182.615,412.401,-85.188,-175.996,9.054,148.666
C01238=1182.612,412.648,-85.224,-175.995,9.057,148.667
C01239=1182.607,412.896,-85.260,-175.995,9.059,148.668
C01240=1182.604,413.144,-85.296,-175.996,9.061,148.668
C01241=1182.600,413.390,-85.331,-175.995,9.063,148.669
C01242=1182.595,413.638,-85.368,-175.996,9.064,148.669
C01243=1182.592,413.885,-85.403,-175.996,9.067,148.670
C01244=1182.588,414.133,-85.439,-175.995,9.069,148.670
C01245=1182.584,414.380,-85.476,-175.996,9.071,148.671
C01246=1182.580,414.627,-85.511,-175.996,9.073,148.671
C01247=1182.576,414.875,-85.547,-175.996,9.074,148.672
C01248=1182.572,415.123,-85.583,-175.996,9.077,148.672
C01249=1182.568,415.369,-85.619,-175.996,9.078,148.673
C01250=1182.564,415.590,-85.651,-175.996,9.080,148.673
C01251=1182.561,415.811,-85.683,-175.996,9.082,148.674
C01252=1182.558,416.033,-85.715,-175.996,9.083,148.674
C01253=1182.557,416.254,-85.747,-175.996,9.085,148.675
C01254=1182.557,416.475,-85.779,-175.996,9.087,148.675
C01255=1182.557,416.695,-85.811,-175.996,9.088,148.675
C01256=1182.559,416.916,-85.842,-175.996,9.090,148.676
C01257=1182.562,417.136,-85.873,-175.996,9.091,148.676
C01258=1182.140,417.137,-85.915,-175.999,9.102,148.680
C01259=1182.138,416.915,-85.884,-175.999,9.101,148.680
C01260=1182.136,416.693,-85.852,-175.999,9.099,148.679
C01261=1182.135,416.471,-85.820,-175.999,9.098,148.679
C01262=1182.136,416.249,-85.788,-175.999,9.096,148.678
C01263=1182.137,416.026,-85.756,-175.999,9.094,148.678
C01264=1182.140,415.803,-85.724,-175.999,9.092,148.677
C01265=1182.143,415.581,-85.691,-175.999,9.091,148.677
C01266=1182.147,415.358,-85.659,-175.999,9.089,148.676
C01267=1182.151,415.111,-85.624,-175.999,9.087,148.676
C01268=1182.154,414.864,-85.587,-175.999,9.085,148.675
C01269=1182.158,414.616,-85.551,-175.999,9.084,148.675
C01270=1182.162,414.369,-85.516,-175.999,9.081,148.674
C01271=1182.167,414.122,-85.479,-175.999,9.080,148.674
C01272=1182.171,413.875,-85.444,-175.999,9.078,148.673
C01273=1182.174,413.627,-85.408,-175.999,9.075,148.673
C01274=1182.179,413.379,-85.372,-175.998,9.074,148.672
C01275=1182.182,413.132,-85.336,-175.999,9.071,148.672
C01276=1182.186,412.885,-85.300,-175.998,9.070,148.671
C01277=1182.190,412.637,-85.264,-175.999,9.068,148.671
C01278=1182.194,412.390,-85.228,-175.998,9.066,148.670
C01279=1182.199,412.143,-85.193,-175.998,9.064,148.670
C01280=1182.202,411.896,-85.156,-175.999,9.061,148.669
C01281=1182.206,411.648,-85.121,-175.998,9.060,148.669
C01282=1182.210,411.400,-85.085,-175.998,9.057,148.668
C01283=1182.214,411.153,-85.049,-175.998,9.056,148.667
C01284=1182.217,410.906,-85.013,-175.998,9.054,148.667
C01285=1182.221,410.658,-84.977,-175.998,9.051,148.666
C01286=1182.225,410.411,-84.941,-175.998,9.050,148.666
C01287=1182.229,410.164,-84.906,-175.998,9.047,148.665
C01288=1182.234,409.916,-84.870,-175.998,9.045,148.665
C01289=1182.237,409.669,-84.834,-175.998,9.044,148.664
C01290=1182.241,409.422,-84.798,-175.998,9.041,148.664
C01291=1182.245,409.174,-84.762,-175.998,9.039,148.663
C01292=1182.249,408.926,-84.726,-175.998,9.037,148.663
C01293=1182.253,408.679,-84.691,-175.997,9.035,148.662
C01294=1182.258,408.432,-84.655,-175.998,9.033,148.661
C01295=1182.261,408.185,-84.619,-175.997,9.031,148.661
C01296=1182.265,407.937,-84.583,-175.997,9.029,148.660
C01297=1182.269,407.690,-84.547,-175.997,9.026,148.660
C01298=1182.273,407.442,-84.512,-175.998,9.024,148.659
C01299=1182.276,407.195,-84.476,-175.997,9.022,148.658
C01300=1182.281,406.947,-84.440,-175.997,9.020,148.658
C01301=1182.285,406.701,-84.404,-175.997,9.018,148.657
C01302=1182.288,406.453,-84.368,-175.997,9.016,148.657
C01303=1182.293,406.205,-84.332,-175.997,9.014,148.656
C01304=1182.296,405.958,-84.297,-175.997,9.012,148.656
C01305=1182.300,405.710,-84.261,-175.997,9.009,148.655
C01306=1182.304,405.462,-84.225,-175.997,9.007,148.654
C01307=1182.309,405.216,-84.190,-175.997,9.005,148.654
C01308=1182.312,404.969,-84.154,-175.997,9.003,148.653
C01309=1182.316,404.721,-84.118,-175.997,9.000,148.653
C01310=1182.320,404.473,-84.082,-175.997,8.998,148.652
C01311=1182.324,404.226,-84.046,-175.997,8.996,148.652
C01312=1182.327,403.978,-84.011,-175.997,8.994,148.651
C01313=1182.332,403.731,-83.975,-175.997,8.992,148.650
C01314=1182.336,403.484,-83.939,-175.997,8.989,148.650
C01315=1182.340,403.236,-83.904,-175.997,8.987,148.649
C01316=1182.343,402.989,-83.868,-175.997,8.985,148.649
C01317=1182.348,402.741,-83.832,-175.997,8.982,148.648
C01318=1182.352,402.495,-83.796,-175.997,8.980,148.647
C01319=1182.355,402.247,-83.761,-175.997,8.977,148.647
C01320=1182.359,402.000,-83.725,-175.997,8.975,148.646
C01321=1182.364,401.752,-83.689,-175.997,8.973,148.645
C01322=1182.367,401.505,-83.654,-175.997,8.971,148.645
C01323=1182.371,401.257,-83.618,-175.997,8.968,148.644
C01324=1182.375,401.010,-83.583,-175.997,8.966,148.644
C01325=1182.380,400.762,-83.547,-175.997,8.964,148.643
C01326=1182.383,400.515,-83.511,-175.997,8.961,148.642
C01327=1182.387,400.267,-83.476,-175.997,8.959,148.642
C01328=1182.391,400.020,-83.440,-175.997,8.956,148.641
C01329=1182.396,399.773,-83.404,-175.997,8.954,148.641
C01330=1182.399,399.525,-83.369,-175.997,8.952,148.640
C01331=1182.403,399.278,-83.333,-175.997,8.949,148.639
C01332=1182.407,399.030,-83.298,-175.997,8.947,148.639
C01333=1182.411,398.782,-83.261,-175.998,8.944,148.638
C01334=1182.415,398.536,-83.226,-175.998,8.941,148.637
C01335=1182.419,398.288,-83.191,-175.998,8.939,148.637
C01336=1182.423,398.041,-83.155,-175.998,8.936,148.636
C01337=1182.427,397.793,-83.119,-175.998,8.934,148.636
C01338=1182.431,397.545,-83.083,-175.998,8.931,148.635
C01339=1182.435,397.299,-83.048,-175.998,8.929,148.634
C01340=1182.438,397.051,-83.013,-175.998,8.927,148.634
C01341=1182.442,396.804,-82.977,-175.998,8.924,148.633
C01342=1182.447,396.556,-82.941,-175.999,8.921,148.632
C01343=1182.451,396.309,-82.906,-175.999,8.919,148.632
C01344=1182.454,396.061,-82.870,-175.999,8.916,148.631
C01345=1182.458,395.814,-82.835,-175.999,8.914,148.631
C01346=1182.462,395.566,-82.799,-175.999,8.911,148.630
C01347=1182.467,395.319,-82.763,-176.000,8.908,148.629
C01348=1182.470,395.072,-82.728,-176.000,8.906,148.629
C01349=1182.474,394.824,-82.692,-176.000,8.903,148.628
C01350=1182.478,394.577,-82.657,-176.000,8.901,148.627
C01351=1182.481,394.329,-82.621,-176.000,8.898,148.627
C01352=1182.486,394.083,-82.586,-176.000,8.895,148.626
C01353=1182.490,393.834,-82.551,-176.001,8.893,148.625
C01354=1182.494,393.587,-82.515,-176.001,8.889,148.625
C01355=1182.498,393.339,-82.480,-176.001,8.887,148.624
C01356=1182.502,393.092,-82.444,-176.001,8.885,148.624
C01357=1182.506,392.845,-82.409,-176.002,8.881,148.623
C01358=1182.509,392.597,-82.373,-176.002,8.879,148.622
C01359=1182.515,392.313,-82.333,-176.002,8.876,148.622
C01360=1182.519,392.030,-82.292,-176.003,8.872,148.621
C01361=1182.523,391.745,-82.251,-176.003,8.869,148.620
C01362=1182.528,391.462,-82.211,-176.003,8.866,148.619
C01363=1182.531,391.214,-82.175,-176.004,8.863,148.619
C01364=1182.535,390.967,-82.140,-176.004,8.861,148.618
C01365=1182.540,390.719,-82.104,-176.005,8.858,148.617
C01366=1182.544,390.471,-82.069,-176.005,8.855,148.617
C01367=1182.548,390.224,-82.033,-176.005,8.852,148.616
C01368=1182.551,389.976,-81.998,-176.006,8.849,148.616
C01369=1182.556,389.730,-81.963,-176.006,8.846,148.615
C01370=1182.559,389.482,-81.927,-176.007,8.843,148.614
C01371=1182.563,389.234,-81.892,-176.007,8.841,148.614
C01372=1182.568,388.987,-81.857,-176.007,8.838,148.613
C01373=1182.571,388.740,-81.822,-176.008,8.834,148.612
C01374=1182.575,388.492,-81.786,-176.008,8.832,148.612
C01375=1182.579,388.244,-81.751,-176.009,8.829,148.611
C01376=1182.584,387.997,-81.715,-176.010,8.826,148.610
C01377=1182.588,387.749,-81.680,-176.010,8.823,148.610
C01378=1182.591,387.502,-81.644,-176.010,8.820,148.609
C01379=1182.596,387.254,-81.610,-176.011,8.817,148.609
C01380=1182.599,387.007,-81.574,-176.012,8.814,148.608
C01381=1182.603,386.759,-81.539,-176.012,8.811,148.607
C01382=1182.607,386.513,-81.504,-176.012,8.808,148.607
C01383=1182.611,386.265,-81.469,-176.013,8.805,148.606
C01384=1182.615,386.017,-81.433,-176.014,8.802,148.606
C01385=1182.619,385.770,-81.398,-176.014,8.799,148.605
C01386=1182.623,385.522,-81.363,-176.015,8.796,148.604
C01387=1182.627,385.275,-81.328,-176.016,8.793,148.604
C01388=1182.631,385.027,-81.292,-176.016,8.790,148.603
C01389=1182.635,384.780,-81.258,-176.017,8.787,148.602
C01390=1182.639,384.532,-81.222,-176.018,8.784,148.602
C01391=1182.642,384.285,-81.186,-176.018,8.781,148.601
C01392=1182.647,384.037,-81.152,-176.019,8.778,148.601
C01393=1182.651,383.790,-81.116,-176.020,8.774,148.600
C01394=1182.655,383.543,-81.081,-176.021,8.771,148.599
C01395=1182.659,383.295,-81.046,-176.022,8.768,148.599
C01396=1182.663,383.047,-81.011,-176.022,8.765,148.598
C01397=1182.667,382.800,-80.976,-176.023,8.762,148.598
C01398=1182.671,382.552,-80.941,-176.024,8.759,148.597
C01399=1182.674,382.305,-80.905,-176.025,8.756,148.596
C01400=1182.679,382.058,-80.871,-176.026,8.752,148.596
C01401=1182.683,381.810,-80.835,-176.027,8.749,148.595
C01402=1182.687,381.562,-80.800,-176.028,8.746,148.595
C01403=1182.691,381.315,-80.765,-176.029,8.743,148.594
C01404=1182.695,381.067,-80.730,-176.030,8.740,148.593
C01405=1182.699,380.820,-80.695,-176.030,8.736,148.593
C01406=1182.703,380.572,-80.660,-176.032,8.733,148.592
C01407=1182.706,380.325,-80.626,-176.033,8.729,148.592
C01408=1182.711,380.077,-80.591,-176.033,8.726,148.591
C01409=1182.714,379.830,-80.555,-176.034,8.723,148.591
C01410=1182.719,379.583,-80.521,-176.036,8.719,148.590
C01411=1182.722,379.335,-80.485,-176.036,8.716,148.589
C01412=1182.726,379.087,-80.451,-176.037,8.713,148.589
C01413=1182.731,378.840,-80.415,-176.038,8.710,148.588
C01414=1182.735,378.592,-80.381,-176.040,8.706,148.588
C01415=1182.739,378.345,-80.345,-176.041,8.703,148.587
C01416=1182.743,378.097,-80.311,-176.042,8.700,148.587
C01417=1182.746,377.850,-80.276,-176.043,8.696,148.586
C01418=1182.750,377.602,-80.241,-176.044,8.694,148.586
C01419=1182.754,377.354,-80.206,-176.046,8.690,148.585
C01420=1182.759,377.108,-80.171,-176.046,8.687,148.584
C01421=1182.763,376.859,-80.136,-176.047,8.683,148.584
C01422=1182.767,376.613,-80.101,-176.049,8.680,148.583
C01423=1182.770,376.365,-80.067,-176.050,8.677,148.583
C01424=1182.774,376.117,-80.032,-176.051,8.673,148.582
C01425=1182.778,375.870,-79.997,-176.052,8.670,148.582
C01426=1182.782,375.622,-79.962,-176.054,8.666,148.581
C01427=1182.787,375.374,-79.928,-176.055,8.663,148.581
C01428=1182.790,375.127,-79.893,-176.056,8.659,148.580
C01429=1182.794,374.880,-79.858,-176.057,8.656,148.579
C01430=1182.798,374.632,-79.823,-176.059,8.653,148.579
C01431=1182.803,374.384,-79.789,-176.060,8.650,148.578
C01432=1182.807,374.137,-79.753,-176.062,8.646,148.578
C01433=1182.810,373.890,-79.719,-176.062,8.643,148.577
C01434=1182.814,373.641,-79.685,-176.064,8.639,148.577
C01435=1182.819,373.395,-79.649,-176.065,8.636,148.576
C01436=1182.823,373.147,-79.615,-176.067,8.632,148.576
C01437=1182.826,372.899,-79.581,-176.068,8.629,148.575
C01438=1182.830,372.651,-79.546,-176.070,8.626,148.575
C01439=1182.835,372.404,-79.511,-176.071,8.622,148.575
C01440=1182.838,372.157,-79.477,-176.073,8.618,148.574
C01441=1182.842,371.909,-79.442,-176.074,8.615,148.573
C01442=1182.846,371.661,-79.407,-176.075,8.612,148.573
C01443=1182.851,371.414,-79.373,-176.077,8.609,148.572
C01444=1182.854,371.166,-79.339,-176.078,8.605,148.572
C01445=1182.859,370.919,-79.304,-176.080,8.601,148.571
C01446=1182.863,370.670,-79.269,-176.082,8.598,148.571
C01447=1182.866,370.424,-79.235,-176.083,8.595,148.571
C01448=1182.870,370.176,-79.200,-176.085,8.591,148.570
C01449=1182.875,369.928,-79.165,-176.086,8.587,148.570
C01450=1182.878,369.681,-79.131,-176.087,8.584,148.569
C01451=1182.883,369.433,-79.097,-176.089,8.581,148.569
C01452=1182.887,369.185,-79.062,-176.091,8.577,148.568
C01453=1182.890,368.938,-79.028,-176.093,8.574,148.568
C01454=1182.895,368.690,-78.993,-176.094,8.570,148.567
C01455=1182.898,368.443,-78.959,-176.095,8.567,148.567
C01456=1182.903,368.195,-78.925,-176.097,8.563,148.566
C01457=1182.907,367.947,-78.890,-176.099,8.560,148.566
C01458=1182.911,367.700,-78.856,-176.101,8.556,148.566
C01459=1182.915,367.452,-78.821,-176.102,8.553,148.565
C01460=1182.918,367.205,-78.787,-176.104,8.550,148.565
C01461=1182.923,366.957,-78.753,-176.106,8.546,148.564
C01462=1182.927,366.709,-78.718,-176.108,8.542,148.564
C01463=1182.931,366.428,-78.679,-176.109,8.539,148.563
C01464=1182.935,366.147,-78.640,-176.111,8.534,148.563
C01465=1182.940,365.864,-78.602,-176.113,8.530,148.562
C01466=1182.945,365.584,-78.563,-176.115,8.527,148.562
C01467=1182.949,365.336,-78.528,-176.117,8.523,148.561
C01468=1182.953,365.088,-78.494,-176.119,8.520,148.561
C01469=1182.957,364.840,-78.460,-176.121,8.516,148.561
C01470=1182.961,364.593,-78.426,-176.123,8.513,148.560
C01471=1182.965,364.346,-78.391,-176.125,8.509,148.560
C01472=1182.969,364.097,-78.358,-176.126,8.505,148.559
C01473=1182.973,363.850,-78.323,-176.128,8.502,148.559
C01474=1182.977,363.603,-78.289,-176.129,8.499,148.559
C01475=1182.981,363.355,-78.255,-176.132,8.496,148.558
C01476=1182.985,363.107,-78.221,-176.133,8.492,148.558
C01477=1182.989,362.860,-78.188,-176.135,8.488,148.558
C01478=1182.993,362.612,-78.153,-176.137,8.485,148.557
C01479=1182.997,362.365,-78.119,-176.139,8.481,148.557
C01480=1183.002,362.117,-78.085,-176.141,8.478,148.556
C01481=1183.005,361.869,-78.051,-176.143,8.474,148.556
C01482=1183.009,361.622,-78.017,-176.145,8.471,148.556
C01483=1183.014,361.374,-77.982,-176.147,8.467,148.555
C01484=1183.017,361.126,-77.949,-176.149,8.464,148.555
C01485=1183.022,360.878,-77.914,-176.151,8.460,148.555
C01486=1183.025,360.631,-77.881,-176.153,8.457,148.554
C01487=1183.029,360.383,-77.847,-176.155,8.453,148.554
C01488=1183.034,360.136,-77.813,-176.157,8.450,148.554
C01489=1183.038,359.888,-77.779,-176.159,8.446,148.553
C01490=1183.042,359.641,-77.746,-176.161,8.443,148.553
C01491=1183.046,359.393,-77.711,-176.163,8.439,148.553
C01492=1183.050,359.145,-77.678,-176.165,8.436,148.552
C01493=1183.053,358.898,-77.644,-176.167,8.432,148.552
C01494=1183.058,358.649,-77.610,-176.169,8.429,148.552
C01495=1183.062,358.402,-77.576,-176.171,8.425,148.551
C01496=1183.066,358.154,-77.543,-176.173,8.422,148.551
C01497=1183.070,357.907,-77.508,-176.175,8.418,148.551
C01498=1183.074,357.658,-77.475,-176.177,8.415,148.550
C01499=1183.078,357.411,-77.441,-176.180,8.412,148.550
C01500=1183.082,357.163,-77.408,-176.181,8.408,148.550
C01501=1183.086,356.916,-77.373,-176.184,8.405,148.550
C01502=1183.091,356.668,-77.340,-176.186,8.401,148.549
C01503=1183.094,356.420,-77.306,-176.188,8.398,148.549
C01504=1183.098,356.173,-77.273,-176.190,8.395,148.549
C01505=1183.103,355.925,-77.239,-176.192,8.391,148.548
C01506=1183.107,355.678,-77.205,-176.194,8.388,148.548
C01507=1183.110,355.429,-77.171,-176.196,8.384,148.548
C01508=1183.114,355.182,-77.138,-176.198,8.381,148.547
C01509=1183.118,354.934,-77.104,-176.200,8.377,148.547
C01510=1183.123,354.686,-77.071,-176.203,8.374,148.547
C01511=1183.127,354.439,-77.037,-176.205,8.370,148.546
C01512=1183.131,354.191,-77.004,-176.207,8.367,148.546
C01513=1183.134,353.943,-76.970,-176.209,8.364,148.546
C01514=1183.139,353.695,-76.937,-176.211,8.360,148.546
C01515=1183.142,353.448,-76.903,-176.213,8.357,148.545
C01516=1183.147,353.200,-76.869,-176.215,8.353,148.545
C01517=1183.151,352.952,-76.836,-176.218,8.350,148.545
C01518=1183.156,352.705,-76.803,-176.220,8.347,148.545
C01519=1183.159,352.458,-76.769,-176.222,8.343,148.544
C01520=1183.163,352.209,-76.736,-176.224,8.340,148.544
C01521=1183.167,351.961,-76.702,-176.226,8.337,148.544
C01522=1183.171,351.714,-76.669,-176.228,8.333,148.544
C01523=1183.175,351.466,-76.636,-176.231,8.330,148.543
C01524=1183.180,351.219,-76.602,-176.233,8.326,148.543
C01525=1183.184,350.971,-76.569,-176.235,8.323,148.543
C01526=1183.188,350.723,-76.535,-176.237,8.320,148.543
C01527=1183.192,350.475,-76.502,-176.239,8.316,148.542
C01528=1183.197,350.228,-76.469,-176.242,8.313,148.542
C01529=1183.200,349.979,-76.436,-176.244,8.310,148.542
C01530=1183.204,349.731,-76.402,-176.246,8.306,148.541
C01531=1183.208,349.484,-76.369,-176.248,8.303,148.541
C01532=1183.212,349.236,-76.336,-176.250,8.300,148.541
C01533=1183.216,348.989,-76.302,-176.253,8.295,148.541
C01534=1183.220,348.741,-76.269,-176.255,8.292,148.540
C01535=1183.225,348.493,-76.236,-176.257,8.289,148.540
C01536=1183.229,348.246,-76.203,-176.260,8.285,148.540
C01537=1183.233,347.998,-76.170,-176.262,8.282,148.540
C01538=1183.237,347.750,-76.136,-176.264,8.279,148.540
C01539=1183.241,347.502,-76.104,-176.267,8.275,148.539
C01540=1183.246,347.254,-76.071,-176.269,8.272,148.539
C01541=1183.250,347.006,-76.038,-176.271,8.269,148.539
C01542=1183.254,346.759,-76.005,-176.273,8.266,148.539
C01543=1183.258,346.511,-75.971,-176.276,8.262,148.539
C01544=1183.261,346.264,-75.939,-176.277,8.259,148.538
C01545=1183.266,346.016,-75.906,-176.280,8.255,148.538
C01546=1183.270,345.768,-75.872,-176.282,8.252,148.538
C01547=1183.274,345.520,-75.839,-176.284,8.249,148.537
C01548=1183.278,345.273,-75.806,-176.286,8.246,148.537
C01549=1183.282,345.024,-75.774,-176.289,8.243,148.537
C01550=1183.287,344.777,-75.741,-176.291,8.240,148.537
C01551=1183.291,344.529,-75.707,-176.293,8.237,148.537
C01552=1183.295,344.281,-75.674,-176.295,8.233,148.537
C01553=1183.298,344.034,-75.642,-176.298,8.230,148.536
C01554=1183.303,343.785,-75.609,-176.300,8.227,148.536
C01555=1183.307,343.538,-75.576,-176.302,8.223,148.536
C01556=1183.311,343.290,-75.543,-176.304,8.220,148.536
C01557=1183.315,343.042,-75.510,-176.307,8.217,148.536
C01558=1183.319,342.794,-75.477,-176.309,8.213,148.535
C01559=1183.323,342.546,-75.445,-176.311,8.210,148.535
C01560=1183.327,342.299,-75.412,-176.313,8.207,148.535
C01561=1183.331,342.050,-75.379,-176.316,8.203,148.535
C01562=1183.336,341.803,-75.346,-176.318,8.200,148.534
C01563=1183.340,341.556,-75.313,-176.321,8.197,148.534
C01564=1183.344,341.308,-75.281,-176.323,8.194,148.534
C01565=1183.348,341.060,-75.248,-176.325,8.190,148.534
C01566=1183.352,340.812,-75.215,-176.327,8.187,148.534
C01567=1183.357,340.533,-75.179,-176.330,8.183,148.534
C01568=1183.362,340.253,-75.142,-176.332,8.180,148.533
C01569=1183.366,339.975,-75.105,-176.335,8.175,148.533
C01570=1183.371,339.696,-75.069,-176.338,8.172,148.533
C01571=1183.375,339.448,-75.036,-176.340,8.169,148.533
C01572=1183.379,339.200,-75.003,-176.343,8.166,148.533
C01573=1183.383,338.953,-74.970,-176.345,8.163,148.532
C01574=1183.388,338.705,-74.938,-176.347,8.159,148.532
C01575=1183.392,338.457,-74.905,-176.350,8.156,148.532
C01576=1183.395,338.209,-74.873,-176.352,8.153,148.532
C01577=1183.400,337.961,-74.841,-176.354,8.150,148.532
C01578=1183.404,337.713,-74.808,-176.357,8.146,148.532
C01579=1183.408,337.465,-74.776,-176.359,8.143,148.531
C01580=1183.412,337.217,-74.743,-176.361,8.140,148.531
C01581=1183.416,336.970,-74.711,-176.364,8.137,148.531
C01582=1183.420,336.722,-74.678,-176.366,8.133,148.531
C01583=1183.425,336.474,-74.646,-176.368,8.130,148.531
C01584=1183.429,336.226,-74.614,-176.371,8.127,148.531
C01585=1183.433,335.978,-74.581,-176.373,8.124,148.530
C01586=1183.436,335.730,-74.549,-176.375,8.120,148.530
C01587=1183.441,335.483,-74.517,-176.378,8.117,148.530
C01588=1183.445,335.235,-74.484,-176.380,8.114,148.530
C01589=1183.449,334.987,-74.452,-176.383,8.111,148.530
C01590=1183.454,334.738,-74.419,-176.385,8.107,148.530
C01591=1183.457,334.491,-74.387,-176.387,8.105,148.530
C01592=1183.462,334.243,-74.355,-176.389,8.102,148.529
C01593=1183.466,333.995,-74.323,-176.392,8.099,148.529
C01594=1183.470,333.747,-74.290,-176.394,8.096,148.529
C01595=1183.474,333.500,-74.258,-176.397,8.092,148.529
C01596=1183.479,333.252,-74.226,-176.399,8.089,148.529
C01597=1183.482,333.004,-74.194,-176.402,8.086,148.529
C01598=1183.487,332.756,-74.161,-176.404,8.083,148.529
C01599=1183.491,332.507,-74.130,-176.406,8.079,148.528
C01600=1183.495,332.261,-74.097,-176.409,8.076,148.528
C01601=1183.499,332.012,-74.065,-176.411,8.073,148.528
C01602=1183.503,331.764,-74.033,-176.413,8.070,148.528
C01603=1183.507,331.516,-74.001,-176.416,8.067,148.528
C01604=1183.511,331.269,-73.969,-176.418,8.063,148.528
C01605=1183.516,331.020,-73.937,-176.421,8.060,148.528
C01606=1183.520,330.772,-73.905,-176.423,8.057,148.528
C01607=1183.524,330.525,-73.873,-176.425,8.054,148.527
C01608=1183.528,330.277,-73.840,-176.428,8.050,148.527
C01609=1183.532,330.029,-73.808,-176.430,8.047,148.527
C01610=1183.537,329.782,-73.776,-176.433,8.044,148.527
C01611=1183.541,329.534,-73.745,-176.435,8.041,148.527
C01612=1183.544,329.285,-73.713,-176.437,8.039,148.527
C01613=1183.549,329.038,-73.681,-176.439,8.035,148.527
C01614=1183.553,328.790,-73.649,-176.442,8.032,148.527
C01615=1183.557,328.542,-73.617,-176.444,8.029,148.526
C01616=1183.562,328.294,-73.585,-176.447,8.026,148.526
C01617=1183.566,328.045,-73.554,-176.449,8.023,148.526
C01618=1183.569,327.797,-73.522,-176.452,8.020,148.526
C01619=1183.575,327.550,-73.490,-176.454,8.016,148.526
C01620=1183.578,327.302,-73.458,-176.457,8.013,148.526
C01621=1183.582,327.054,-73.426,-176.459,8.010,148.526
C01622=1183.586,326.806,-73.395,-176.462,8.007,148.526
C01623=1183.591,326.558,-73.362,-176.464,8.004,148.526
C01624=1183.594,326.310,-73.330,-176.466,8.000,148.525
C01625=1183.599,326.063,-73.299,-176.469,7.997,148.525
C01626=1183.603,325.814,-73.268,-176.471,7.994,148.525
C01627=1183.608,325.566,-73.236,-176.474,7.992,148.525
C01628=1183.611,325.318,-73.204,-176.476,7.989,148.525
C01629=1183.615,325.070,-73.172,-176.479,7.986,148.525
C01630=1183.619,324.823,-73.140,-176.481,7.982,148.525
C01631=1183.623,324.574,-73.109,-176.484,7.979,148.525
C01632=1183.629,324.327,-73.077,-176.486,7.976,148.525
C01633=1183.632,324.079,-73.045,-176.489,7.973,148.525
C01634=1183.636,323.830,-73.014,-176.491,7.970,148.524
C01635=1183.641,323.583,-72.983,-176.493,7.967,148.524
C01636=1183.644,323.334,-72.951,-176.496,7.963,148.524
C01637=1183.649,323.087,-72.920,-176.498,7.960,148.524
C01638=1183.653,322.838,-72.888,-176.501,7.957,148.524
C01639=1183.658,322.591,-72.856,-176.503,7.954,148.524
C01640=1183.661,322.343,-72.824,-176.505,7.952,148.524
C01641=1183.666,322.095,-72.794,-176.508,7.949,148.524
C01642=1183.670,321.847,-72.762,-176.510,7.945,148.524
C01643=1183.674,321.599,-72.730,-176.513,7.942,148.524
C01644=1183.678,321.351,-72.699,-176.516,7.939,148.524
C01645=1183.682,321.103,-72.667,-176.518,7.936,148.523
C01646=1183.686,320.855,-72.637,-176.520,7.933,148.523
C01647=1183.690,320.607,-72.605,-176.523,7.930,148.523
C01648=1183.695,320.359,-72.574,-176.525,7.927,148.523
C01649=1183.698,320.111,-72.542,-176.528,7.923,148.523
C01650=1183.703,319.863,-72.511,-176.530,7.920,148.523
C01651=1183.707,319.614,-72.479,-176.533,7.918,148.523
C01652=1183.712,319.367,-72.448,-176.535,7.915,148.523
C01653=1183.716,319.118,-72.416,-176.538,7.912,148.523
C01654=1183.720,318.871,-72.386,-176.540,7.908,148.523
C01655=1183.725,318.623,-72.354,-176.543,7.905,148.523
C01656=1183.729,318.375,-72.323,-176.545,7.902,148.523
C01657=1183.732,318.128,-72.292,-176.547,7.899,148.523
C01658=1183.736,317.879,-72.261,-176.550,7.896,148.523
C01659=1183.741,317.631,-72.230,-176.552,7.893,148.522
C01660=1183.745,317.383,-72.198,-176.555,7.890,148.522
C01661=1183.749,317.135,-72.168,-176.558,7.887,148.522
C01662=1183.753,316.887,-72.136,-176.560,7.884,148.522
C01663=1183.757,316.639,-72.105,-176.562,7.881,148.522
C01664=1183.762,316.391,-72.074,-176.565,7.878,148.522
C01665=1183.766,316.143,-72.042,-176.567,7.875,148.522
C01666=1183.770,315.895,-72.012,-176.570,7.872,148.522
C01667=1183.774,315.646,-71.980,-176.572,7.869,148.522
C01668=1183.779,315.398,-71.950,-176.575,7.866,148.522
C01669=1183.783,315.151,-71.918,-176.578,7.863,148.522
C01670=1183.787,314.903,-71.888,-176.580,7.859,148.522
C01671=1183.792,314.626,-71.852,-176.583,7.856,148.522
C01672=1183.797,314.349,-71.819,-176.585,7.853,148.522
C01673=1183.802,314.073,-71.784,-176.588,7.849,148.521
C01674=1183.806,313.796,-71.749,-176.591,7.846,148.521
C01675=1183.810,313.548,-71.718,-176.594,7.843,148.521
C01676=1183.814,313.299,-71.687,-176.596,7.840,148.521
C01677=1183.818,313.052,-71.657,-176.599,7.837,148.521
C01678=1183.823,312.804,-71.626,-176.601,7.835,148.521
C01679=1183.827,312.556,-71.594,-176.603,7.832,148.521
C01680=1183.831,312.308,-71.564,-176.606,7.828,148.521
C01681=1183.836,312.060,-71.533,-176.608,7.825,148.521
C01682=1183.839,311.812,-71.502,-176.611,7.822,148.521
C01683=1183.844,311.564,-71.472,-176.613,7.819,148.521
C01684=1183.848,311.316,-71.441,-176.616,7.816,148.521
C01685=1183.853,311.068,-71.410,-176.619,7.813,148.521
C01686=1183.856,310.819,-71.379,-176.621,7.811,148.521
C01687=1183.861,310.571,-71.349,-176.623,7.808,148.521
C01688=1183.865,310.323,-71.318,-176.626,7.805,148.521
C01689=1183.869,310.075,-71.287,-176.629,7.802,148.521
C01690=1183.873,309.827,-71.257,-176.631,7.798,148.521
C01691=1183.878,309.579,-71.226,-176.634,7.795,148.521
C01692=1183.882,309.330,-71.195,-176.636,7.792,148.521
C01693=1183.886,309.083,-71.165,-176.638,7.790,148.521
C01694=1183.890,308.835,-71.134,-176.641,7.787,148.521
C01695=1183.895,308.587,-71.103,-176.643,7.784,148.521
C01696=1183.898,308.339,-71.073,-176.646,7.781,148.521
C01697=1183.903,308.091,-71.042,-176.648,7.778,148.520
C01698=1183.908,307.842,-71.012,-176.651,7.775,148.520
C01699=1183.912,307.594,-70.982,-176.654,7.772,148.520
C01700=1183.916,307.346,-70.950,-176.656,7.769,148.521
C01701=1183.920,307.098,-70.920,-176.658,7.766,148.520
C01702=1183.924,306.850,-70.889,-176.661,7.763,148.520
C01703=1183.929,306.602,-70.859,-176.664,7.760,148.520
C01704=1183.933,306.355,-70.829,-176.666,7.757,148.520
C01705=1183.937,306.105,-70.798,-176.669,7.754,148.520
C01706=1183.941,305.858,-70.768,-176.671,7.751,148.520
C01707=1183.945,305.610,-70.737,-176.674,7.749,148.520
C01708=1183.950,305.362,-70.706,-176.676,7.746,148.520
C01709=1183.954,305.113,-70.677,-176.679,7.743,148.520
C01710=1183.958,304.865,-70.646,-176.681,7.739,148.520
C01711=1183.962,304.617,-70.616,-176.684,7.736,148.520
C01712=1183.967,304.369,-70.586,-176.687,7.733,148.520
C01713=1183.971,304.121,-70.555,-176.689,7.730,148.520
C01714=1183.976,303.873,-70.525,-176.691,7.728,148.520
C01715=1183.980,303.625,-70.495,-176.694,7.725,148.520
C01716=1183.984,303.377,-70.464,-176.697,7.722,148.520
C01717=1183.988,303.128,-70.434,-176.699,7.719,148.520
C01718=1183.993,302.880,-70.404,-176.702,7.716,148.520
C01719=1183.996,302.632,-70.374,-176.704,7.712,148.520
C01720=1184.001,302.384,-70.343,-176.706,7.710,148.520
C01721=1184.005,302.136,-70.313,-176.709,7.707,148.520
C01722=1184.010,301.888,-70.283,-176.712,7.704,148.520
C01723=1184.014,301.640,-70.253,-176.715,7.701,148.520
C01724=1184.017,301.391,-70.223,-176.717,7.698,148.520
C01725=1184.022,301.143,-70.193,-176.720,7.695,148.520
C01726=1184.026,300.895,-70.163,-176.722,7.693,148.520
C01727=1184.031,300.647,-70.132,-176.724,7.690,148.520
C01728=1184.035,300.399,-70.102,-176.727,7.687,148.520
C01729=1184.039,300.151,-70.073,-176.730,7.684,148.520
C01730=1184.044,299.903,-70.042,-176.733,7.681,148.520
C01731=1184.048,299.654,-70.013,-176.734,7.678,148.520
C01732=1184.052,299.406,-69.982,-176.737,7.675,148.520
C01733=1184.057,299.158,-69.952,-176.740,7.672,148.520
C01734=1184.061,298.911,-69.922,-176.742,7.669,148.520
C01735=1184.065,298.662,-69.892,-176.745,7.666,148.520
C01736=1184.069,298.413,-69.862,-176.748,7.663,148.520
C01737=1184.073,298.165,-69.832,-176.750,7.661,148.520
C01738=1184.078,297.917,-69.802,-176.752,7.658,148.520
C01739=1184.082,297.668,-69.773,-176.755,7.655,148.520
C01740=1184.086,297.421,-69.743,-176.758,7.652,148.520
C01741=1184.090,297.173,-69.713,-176.760,7.649,148.520
C01742=1184.095,296.924,-69.683,-176.763,7.647,148.520
C01743=1184.099,296.676,-69.653,-176.765,7.644,148.520
C01744=1184.103,296.428,-69.623,-176.768,7.641,148.520
C01745=1184.107,296.180,-69.594,-176.770,7.637,148.520
C01746=1184.112,295.932,-69.563,-176.773,7.634,148.520
C01747=1184.116,295.684,-69.534,-176.775,7.632,148.520
C01748=1184.120,295.435,-69.504,-176.778,7.629,148.520
C01749=1184.124,295.187,-69.475,-176.781,7.626,148.520
C01750=1184.129,294.939,-69.445,-176.783,7.623,148.520
C01751=1184.133,294.691,-69.415,-176.786,7.620,148.520
C01752=1184.137,294.443,-69.385,-176.788,7.618,148.520
C01753=1184.142,294.194,-69.356,-176.791,7.615,148.520
C01754=1184.146,293.946,-69.326,-176.793,7.612,148.520
C01755=1184.150,293.698,-69.297,-176.796,7.609,148.520
C01756=1184.154,293.449,-69.267,-176.799,7.606,148.520
C01757=1184.159,293.202,-69.237,-176.801,7.604,148.520
C01758=1184.163,292.953,-69.207,-176.803,7.601,148.520
C01759=1184.167,292.705,-69.178,-176.806,7.598,148.520
C01760=1184.172,292.457,-69.149,-176.809,7.595,148.520
C01761=1184.176,292.209,-69.119,-176.812,7.592,148.520
C01762=1184.180,291.961,-69.090,-176.814,7.590,148.520
C01763=1184.184,291.713,-69.060,-176.816,7.587,148.520
C01764=1184.189,291.464,-69.031,-176.819,7.584,148.520
C01765=1184.193,291.216,-69.001,-176.822,7.581,148.520
C01766=1184.198,290.968,-68.971,-176.824,7.578,148.520
C01767=1184.202,290.719,-68.942,-176.826,7.575,148.520
C01768=1184.206,290.471,-68.912,-176.829,7.572,148.520
C01769=1184.210,290.223,-68.883,-176.832,7.569,148.520
C01770=1184.214,289.974,-68.853,-176.834,7.567,148.520
C01771=1184.219,289.727,-68.824,-176.837,7.564,148.520
C01772=1184.223,289.479,-68.795,-176.839,7.561,148.520
C01773=1184.228,289.230,-68.765,-176.842,7.558,148.520
C01774=1184.232,288.982,-68.736,-176.845,7.555,148.520
C01775=1184.236,288.707,-68.704,-176.848,7.552,148.521
C01776=1184.241,288.432,-68.672,-176.850,7.549,148.521
C01777=1184.245,288.158,-68.639,-176.853,7.546,148.521
C01778=1184.251,287.883,-68.607,-176.856,7.543,148.521
C01779=1184.255,287.635,-68.577,-176.858,7.540,148.521
C01780=1184.259,287.387,-68.548,-176.861,7.537,148.521
C01781=1184.264,287.139,-68.519,-176.863,7.535,148.521
C01782=1184.269,286.890,-68.490,-176.866,7.532,148.521
C01783=1184.273,286.642,-68.461,-176.869,7.529,148.521
C01784=1184.276,286.394,-68.432,-176.871,7.526,148.521
C01785=1184.280,286.146,-68.402,-176.874,7.524,148.521
C01786=1184.285,285.897,-68.374,-176.876,7.521,148.521
C01787=1184.290,285.649,-68.345,-176.879,7.518,148.521
C01788=1184.294,285.401,-68.315,-176.882,7.515,148.521
C01789=1184.298,285.153,-68.286,-176.884,7.513,148.521
C01790=1184.302,284.904,-68.257,-176.887,7.510,148.521
C01791=1184.307,284.656,-68.228,-176.889,7.507,148.521
C01792=1184.311,284.408,-68.198,-176.892,7.504,148.521
C01793=1184.315,284.159,-68.170,-176.894,7.501,148.521
C01794=1184.319,283.911,-68.141,-176.897,7.498,148.521
C01795=1184.324,283.663,-68.111,-176.900,7.495,148.521
C01796=1184.329,283.415,-68.083,-176.902,7.492,148.521
C01797=1184.333,283.166,-68.053,-176.905,7.490,148.521
C01798=1184.337,282.918,-68.025,-176.907,7.487,148.521
C01799=1184.341,282.670,-67.996,-176.910,7.484,148.522
C01800=1184.346,282.421,-67.967,-176.913,7.481,148.522
C01801=1184.350,282.173,-67.938,-176.915,7.479,148.522
C01802=1184.354,281.925,-67.909,-176.918,7.476,148.522
C01803=1184.359,281.677,-67.880,-176.920,7.473,148.522
C01804=1184.363,281.429,-67.851,-176.923,7.471,148.522
C01805=1184.367,281.180,-67.823,-176.925,7.468,148.522
C01806=1184.372,280.932,-67.794,-176.928,7.465,148.522
C01807=1184.376,280.684,-67.765,-176.931,7.462,148.522
C01808=1184.380,280.435,-67.737,-176.933,7.460,148.522
C01809=1184.384,280.187,-67.707,-176.936,7.457,148.522
